KUKA KRL program: EPS_2_251491_MH05A_A_20251118025200.src

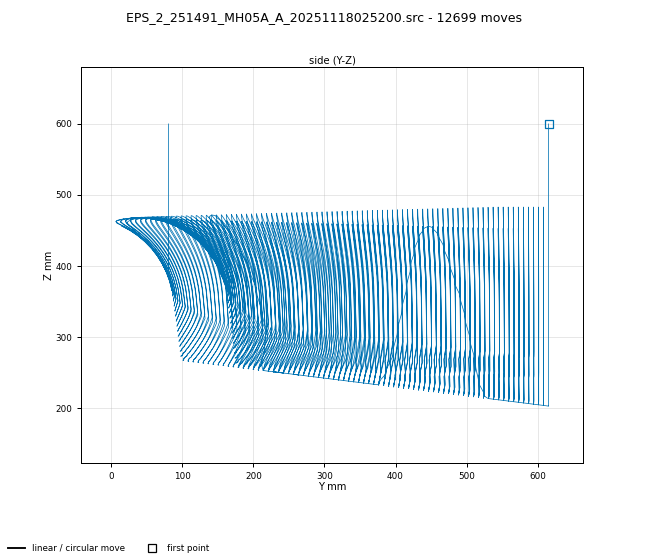
[picture p0: tool path of EPS_2_251491_MH05A_A_20251118025200.src, 12699 of 12701 moves have a stored position in this frame; points joined in program order, loops and branches not executed]
&ACCESS RVP
&REL 4
&COMMENT QRS 19112012
&PARAM EDITMASK = *
DEF PART()
EXT BAS (BAS_COMMAND :IN,REAL :IN )
INT I
BAS (#INITMOV,0 )

;KUKA QRS Post kuka4.cps  Date:22-06-2017 !

File_ID=2922

QRS_PRE_INIT()

;Init var - Until changes are made in qrs_pre_init
Outlet_Square_prg=0
Inlet_1_Square_prg=0
Inlet_2_Square_prg=0
Inlet_3_Square_prg=0
Inlet_4_Square_prg=0
Inlet_5_Square_prg=0

Outlet_1={X 0.000, Y 540.910, Z 382.500, B 0.000, E1 0.000 }
Inlet_1={X 0.000, Y 543.050, Z 352.500, B 0.000, E1 155.000 }
Outlet_1_type=201
Inlet_1_type=201
;QRS#1=Sidecore dimensions
;QRS#2=200-8" PVC SDR 35
;QRS#3=200-8" PVC SDR 35
;QRS#4=
;QRS#5=
;QRS#6=
;QRS#7=
;QRS#8=
;QRS#9=12-08 PSX
;QRS#10=12-08 PSX
;QRS#11=
;QRS#12=
;QRS#13=
;QRS#14=
;QRS#15=
;QRS#16=1220x127x762 2,5'
;QRS#17=EPS Height
;QRS#18=483
;QRS#19=*
;QRS#20= UPDATED VERSION 22-06-2017
;QRS#21=*
Outlet_Square=0100
Inlet_1_Square=0100
Inlet_2_Square=0
Inlet_3_Square=0
Inlet_4_Square=0
Inlet_5_Square=0
Mill_Square=1
Outlet_Square_Prg=204
Inlet_1_Square_prg=204

QRS_INIT()

$ADVANCE=5

; T1
PTP {E1 173.607,E2 173.607}
PTP {X 0,Y 615.506,A -85,B 0,C 180,E1 173.607,E2 173.607,E3 0,E4 0,E5 0,E6 0}
QRS_SPEED_INIT()
LIN {X 0,Y 615.506,Z 600,A -85,B 0,C 180,E1 173.607,E2 173.607,E3 0,E4 0,E5 0,E6 0} C_VEL
LIN {X 0,Y 615.506,Z 212.868,A -85,B 0,C 180,E1 173.607,E2 173.607} C_VEL
LIN {X 0,Y 615.506,Z 204.696,A -85,B 0,C 180,E1 173.607,E2 173.607} C_VEL
LIN {X 0,Y 615.486,Z 202.696,A -85,B 0,C 180,E1 173.421,E2 173.421} C_VEL
LIN {X 0,Y 615.466,Z 202.693,A -85,B 0,C 180,E1 170.801,E2 170.801} C_VEL
LIN {X 0,Y 615.486,Z 202.683,A -85,B 0,C 180,E1 168.139,E2 168.139} C_VEL
LIN {X 0,Y 615.489,Z 202.697,A -85,B 0,C 180,E1 165.451,E2 165.451} C_VEL
LIN {X 0,Y 615.458,Z 202.692,A -85,B 0,C 180,E1 162.729,E2 162.729} C_VEL
LIN {X 0,Y 615.489,Z 202.685,A -85,B 0,C 180,E1 159.967,E2 159.967} C_VEL
LIN {X 0,Y 615.474,Z 202.697,A -85,B 0,C 180,E1 157.155,E2 157.155} C_VEL
LIN {X 0,Y 615.46,Z 202.688,A -85,B 0,C 180,E1 154.436,E2 154.436} C_VEL
LIN {X 0,Y 615.493,Z 202.698,A -85,B 0,C 180,E1 151.548,E2 151.548} C_VEL
LIN {X 0,Y 615.453,Z 202.694,A -85,B 0,C 180,E1 148.919,E2 148.919} C_VEL
LIN {X 0,Y 615.455,Z 202.689,A -85,B 0,C 180,E1 146.47,E2 146.47} C_VEL
LIN {X 0,Y 615.485,Z 202.701,A -85,B 0,C 180,E1 143.575,E2 143.575} C_VEL
LIN {X 0,Y 615.448,Z 202.694,A -85,B 0,C 180,E1 140.942,E2 140.942} C_VEL
LIN {X 0,Y 615.45,Z 202.691,A -85,B 0,C 180,E1 138.523,E2 138.523} C_VEL
LIN {X 0,Y 615.494,Z 202.692,A -85,B 0,C 180,E1 135.851,E2 135.851} C_VEL
LIN {X 0,Y 615.475,Z 202.799,A -85,B 0,C 180,E1 134.199,E2 134.199} C_VEL
LIN {X 0,Y 615.458,Z 220.552,A -85,B 0,C 180,E1 131.282,E2 131.282} C_VEL
LIN {X 0,Y 615.437,Z 235.196,A -85,B 0,C 180,E1 128.908,E2 128.908} C_VEL
LIN {X 0,Y 615.496,Z 241.943,A -85,B 0,C 180,E1 127.817,E2 127.817} C_VEL
LIN {X 0,Y 615.443,Z 348.397,A -85,B 0,C 180,E1 126.553,E2 126.553} C_VEL
LIN {X 0,Y 615.464,Z 361.176,A -85,B 0,C 180,E1 126.278,E2 126.278} C_VEL
LIN {X 0,Y 615.498,Z 372.847,A -85,B 0,C 180,E1 125.908,E2 125.908} C_VEL
LIN {X 0,Y 615.47,Z 385.467,A -85,B 0,C 180,E1 125.366,E2 125.366} C_VEL
LIN {X 0,Y 615.47,Z 397.289,A -85,B 0,C 180,E1 124.698,E2 124.698} C_VEL
LIN {X 0,Y 615.497,Z 408.415,A -85,B 0,C 180,E1 123.899,E2 123.899} C_VEL
LIN {X 0,Y 615.497,Z 418.039,A -85,B 0,C 180,E1 123.04,E2 123.04} C_VEL
LIN {X 0,Y 615.496,Z 427.301,A -85,B 0,C 180,E1 122.008,E2 122.008} C_VEL
LIN {X 0,Y 615.495,Z 433.964,A -85,B 0,C 180,E1 121.087,E2 121.087} C_VEL
LIN {X 0,Y 615.499,Z 439.406,A -85,B 0,C 180,E1 120.159,E2 120.159} C_VEL
LIN {X 0,Y 615.497,Z 444.591,A -85,B 0,C 180,E1 119.031,E2 119.031} C_VEL
LIN {X 0,Y 615.492,Z 448.32,A -85,B 0,C 180,E1 117.915,E2 117.915} C_VEL
LIN {X 0,Y 615.499,Z 450.383,A -85,B 0,C 180,E1 117.046,E2 117.046} C_VEL
LIN {X 0,Y 615.495,Z 451.368,A -85,B 0,C 180,E1 116.444,E2 116.444} C_VEL
LIN {X 0,Y 615.496,Z 452.202,A -85,B 0,C 180,E1 115.57,E2 115.57} C_VEL
LIN {X 0,Y 615.496,Z 452.385,A -85,B 0,C 180,E1 114.991,E2 114.991} C_VEL
LIN {X 0,Y 615.496,Z 451.968,A -85,B 0,C 180,E1 114.009,E2 114.009} C_VEL
LIN {X 0,Y 615.494,Z 450.344,A -85,B 0,C 180,E1 112.844,E2 112.844} C_VEL
LIN {X 0,Y 615.496,Z 447.723,A -85,B 0,C 180,E1 111.783,E2 111.783} C_VEL
LIN {X 0,Y 615.497,Z 443.247,A -85,B 0,C 180,E1 110.558,E2 110.558} C_VEL
LIN {X 0,Y 615.495,Z 437.135,A -85,B 0,C 180,E1 109.338,E2 109.338} C_VEL
LIN {X 0,Y 615.498,Z 430.192,A -85,B 0,C 180,E1 108.281,E2 108.281} C_VEL
LIN {X 0,Y 615.498,Z 421.883,A -85,B 0,C 180,E1 107.27,E2 107.27} C_VEL
LIN {X 0,Y 615.497,Z 413.422,A -85,B 0,C 180,E1 106.433,E2 106.433} C_VEL
LIN {X 0,Y 615.495,Z 403.695,A -85,B 0,C 180,E1 105.65,E2 105.65} C_VEL
LIN {X 0,Y 615.46,Z 393.363,A -85,B 0,C 180,E1 104.973,E2 104.973} C_VEL
LIN {X 0,Y 615.476,Z 382.334,A -85,B 0,C 180,E1 104.395,E2 104.395} C_VEL
LIN {X 0,Y 615.49,Z 370.965,A -85,B 0,C 180,E1 103.932,E2 103.932} C_VEL
LIN {X 0,Y 615.448,Z 359.278,A -85,B 0,C 180,E1 103.58,E2 103.58} C_VEL
LIN {X 0,Y 615.432,Z 346.392,A -85,B 0,C 180,E1 103.328,E2 103.328} C_VEL
LIN {X 0,Y 615.495,Z 241.928,A -85,B 0,C 180,E1 102.091,E2 102.091} C_VEL
LIN {X 0,Y 615.436,Z 225.089,A -85,B 0,C 180,E1 99.365,E2 99.365} C_VEL
LIN {X 0,Y 615.432,Z 210.936,A -85,B 0,C 180,E1 97.052,E2 97.052} C_VEL
LIN {X 0,Y 615.459,Z 202.692,A -85,B 0,C 180,E1 95.673,E2 95.673} C_VEL
LIN {X 0,Y 615.436,Z 202.694,A -85,B 0,C 180,E1 93.273,E2 93.273} C_VEL
LIN {X 0,Y 615.438,Z 202.693,A -85,B 0,C 180,E1 91.309,E2 91.309} C_VEL
LIN {X 0,Y 615.457,Z 202.698,A -85,B 0,C 180,E1 88.691,E2 88.691} C_VEL
LIN {X 0,Y 615.491,Z 202.692,A -85,B 0,C 180,E1 86.072,E2 86.072} C_VEL
LIN {X 0,Y 615.446,Z 202.692,A -85,B 0,C 180,E1 83.443,E2 83.443} C_VEL
LIN {X 0,Y 615.447,Z 202.691,A -85,B 0,C 180,E1 81.463,E2 81.463} C_VEL
LIN {X 0,Y 615.443,Z 202.694,A -85,B 0,C 180,E1 79.135,E2 79.135} C_VEL
LIN {X 0,Y 615.459,Z 202.697,A -85,B 0,C 180,E1 76.798,E2 76.798} C_VEL
LIN {X 0,Y 615.494,Z 202.689,A -85,B 0,C 180,E1 74.095,E2 74.095} C_VEL
LIN {X 0,Y 615.448,Z 202.691,A -85,B 0,C 180,E1 71.353,E2 71.353} C_VEL
LIN {X 0,Y 615.49,Z 202.699,A -85,B 0,C 180,E1 68.568,E2 68.568} C_VEL
LIN {X 0,Y 615.47,Z 202.687,A -85,B 0,C 180,E1 65.728,E2 65.728} C_VEL
LIN {X 0,Y 615.458,Z 202.689,A -85,B 0,C 180,E1 63.555,E2 63.555} C_VEL
LIN {X 0,Y 615.45,Z 202.691,A -85,B 0,C 180,E1 61.34,E2 61.34} C_VEL
LIN {X 0,Y 615.465,Z 202.696,A -85,B 0,C 180,E1 58.918,E2 58.918} C_VEL
LIN {X 0,Y 615.492,Z 202.684,A -85,B 0,C 180,E1 55.979,E2 55.979} C_VEL
LIN {X 0,Y 615.461,Z 202.688,A -85,B 0,C 180,E1 53.574,E2 53.574} C_VEL
LIN {X 0,Y 615.469,Z 202.696,A -85,B 0,C 180,E1 50.94,E2 50.94} C_VEL
LIN {X 0,Y 615.495,Z 202.697,A -85,B 0,C 180,E1 48.527,E2 48.527} C_VEL
LIN {X 0,Y 615.484,Z 202.684,A -85,B 0,C 180,E1 45.851,E2 45.851} C_VEL
LIN {X 0,Y 615.468,Z 202.695,A -85,B 0,C 180,E1 43.046,E2 43.046} C_VEL
LIN {X 0,Y 615.495,Z 202.684,A -85,B 0,C 180,E1 40.09,E2 40.09} C_VEL
LIN {X 0,Y 615.463,Z 202.692,A -85,B 0,C 180,E1 37.244,E2 37.244} C_VEL
LIN {X 0,Y 615.491,Z 202.701,A -85,B 0,C 180,E1 34.702,E2 34.702} C_VEL
LIN {X 0,Y 615.473,Z 202.685,A -85,B 0,C 180,E1 31.686,E2 31.686} C_VEL
LIN {X 0,Y 615.465,Z 202.69,A -85,B 0,C 180,E1 29.408,E2 29.408} C_VEL
LIN {X 0,Y 615.478,Z 202.696,A -85,B 0,C 180,E1 27.044,E2 27.044} C_VEL
LIN {X 0,Y 615.486,Z 202.687,A -85,B 0,C 180,E1 24.272,E2 24.272} C_VEL
LIN {X 0,Y 615.469,Z 202.69,A -85,B 0,C 180,E1 21.433,E2 21.433} C_VEL
LIN {X 0,Y 615.484,Z 202.695,A -85,B 0,C 180,E1 18.605,E2 18.605} C_VEL
LIN {X 0,Y 615.486,Z 202.682,A -85,B 0,C 180,E1 15.905,E2 15.905} C_VEL
LIN {X 0,Y 615.477,Z 202.694,A -85,B 0,C 180,E1 13.202,E2 13.202} C_VEL
LIN {X 0,Y 615.481,Z 202.691,A -85,B 0,C 180,E1 10.527,E2 10.527} C_VEL
LIN {X 0,Y 615.487,Z 202.682,A -85,B 0,C 180,E1 7.876,E2 7.876} C_VEL
LIN {X 0,Y 615.48,Z 202.694,A -85,B 0,C 180,E1 5.241,E2 5.241} C_VEL
LIN {X 0,Y 615.48,Z 202.693,A -85,B 0,C 180,E1 2.618,E2 2.618} C_VEL
LIN {X 0,Y 615.486,Z 202.682,A -85,B 0,C 180,E1 0,E2 0} C_VEL
LIN {X 0,Y 615.479,Z 202.692,A -85,B 0,C 180,E1 -2.618,E2 -2.618} C_VEL
LIN {X 0,Y 615.481,Z 202.695,A -85,B 0,C 180,E1 -5.241,E2 -5.241} C_VEL
LIN {X 0,Y 615.487,Z 202.682,A -85,B 0,C 180,E1 -7.876,E2 -7.876} C_VEL
LIN {X 0,Y 615.48,Z 202.691,A -85,B 0,C 180,E1 -10.527,E2 -10.527} C_VEL
LIN {X 0,Y 615.479,Z 202.695,A -85,B 0,C 180,E1 -13.201,E2 -13.201} C_VEL
LIN {X 0,Y 615.486,Z 202.682,A -85,B 0,C 180,E1 -15.905,E2 -15.905} C_VEL
LIN {X 0,Y 615.486,Z 202.695,A -85,B 0,C 180,E1 -18.646,E2 -18.646} C_VEL
LIN {X 0,Y 615.47,Z 202.69,A -85,B 0,C 180,E1 -21.433,E2 -21.433} C_VEL
LIN {X 0,Y 615.485,Z 202.687,A -85,B 0,C 180,E1 -24.272,E2 -24.272} C_VEL
LIN {X 0,Y 615.473,Z 202.694,A -85,B 0,C 180,E1 -27.178,E2 -27.178} C_VEL
LIN {X 0,Y 615.481,Z 202.683,A -85,B 0,C 180,E1 -29.794,E2 -29.794} C_VEL
LIN {X 0,Y 615.486,Z 202.692,A -85,B 0,C 180,E1 -32.458,E2 -32.458} C_VEL
LIN {X 0,Y 615.494,Z 202.699,A -85,B 0,C 180,E1 -34.815,E2 -34.815} C_VEL
LIN {X 0,Y 615.465,Z 202.692,A -85,B 0,C 180,E1 -37.244,E2 -37.244} C_VEL
LIN {X 0,Y 615.495,Z 202.683,A -85,B 0,C 180,E1 -40.09,E2 -40.09} C_VEL
LIN {X 0,Y 615.47,Z 202.695,A -85,B 0,C 180,E1 -43.046,E2 -43.046} C_VEL
LIN {X 0,Y 615.484,Z 202.683,A -85,B 0,C 180,E1 -45.851,E2 -45.851} C_VEL
LIN {X 0,Y 615.49,Z 202.697,A -85,B 0,C 180,E1 -48.527,E2 -48.527} C_VEL
LIN {X 0,Y 615.462,Z 202.694,A -85,B 0,C 180,E1 -51.094,E2 -51.094} C_VEL
LIN {X 0,Y 615.463,Z 202.688,A -85,B 0,C 180,E1 -53.574,E2 -53.574} C_VEL
LIN {X 0,Y 615.49,Z 202.697,A -85,B 0,C 180,E1 -56.466,E2 -56.466} C_VEL
LIN {X 0,Y 615.458,Z 202.694,A -85,B 0,C 180,E1 -59.079,E2 -59.079} C_VEL
LIN {X 0,Y 615.46,Z 202.688,A -85,B 0,C 180,E1 -61.555,E2 -61.555} C_VEL
LIN {X 0,Y 615.495,Z 202.697,A -85,B 0,C 180,E1 -64.43,E2 -64.43} C_VEL
LIN {X 0,Y 615.451,Z 202.693,A -85,B 0,C 180,E1 -67.154,E2 -67.154} C_VEL
LIN {X 0,Y 615.481,Z 202.766,A -85,B 0,C 180,E1 -67.838,E2 -67.838} C_VEL
LIN {X 0,Y 615.467,Z 223.079,A -85,B 0,C 180,E1 -70.662,E2 -70.662} C_VEL
LIN {X 0,Y 615.458,Z 241.932,A -85,B 0,C 180,E1 -73.242,E2 -73.242} C_VEL
LIN {X 0,Y 615.495,Z 263.272,A -85,B 0,C 180,E1 -76.126,E2 -76.126} C_VEL
LIN {X 0,Y 615.46,Z 270.646,A -85,B 0,C 180,E1 -77.113,E2 -77.113} C_VEL
LIN {X 0,Y 615.467,Z 378.845,A -85,B 0,C 180,E1 -78.41,E2 -78.41} C_VEL
LIN {X 0,Y 615.463,Z 391.355,A -85,B 0,C 180,E1 -78.682,E2 -78.682} C_VEL
LIN {X 0,Y 615.484,Z 404.665,A -85,B 0,C 180,E1 -79.115,E2 -79.115} C_VEL
LIN {X 0,Y 615.486,Z 416.481,A -85,B 0,C 180,E1 -79.64,E2 -79.64} C_VEL
LIN {X 0,Y 615.492,Z 427.997,A -85,B 0,C 180,E1 -80.304,E2 -80.304} C_VEL
LIN {X 0,Y 615.499,Z 438.343,A -85,B 0,C 180,E1 -81.05,E2 -81.05} C_VEL
LIN {X 0,Y 615.497,Z 446.813,A -85,B 0,C 180,E1 -81.794,E2 -81.794} C_VEL
LIN {X 0,Y 615.498,Z 454.607,A -85,B 0,C 180,E1 -82.62,E2 -82.62} C_VEL
LIN {X 0,Y 615.496,Z 462.204,A -85,B 0,C 180,E1 -83.608,E2 -83.608} C_VEL
LIN {X 0,Y 615.498,Z 469.205,A -85,B 0,C 180,E1 -84.759,E2 -84.759} C_VEL
LIN {X 0,Y 615.494,Z 473.852,A -85,B 0,C 180,E1 -85.744,E2 -85.744} C_VEL
LIN {X 0,Y 615.494,Z 477.399,A -85,B 0,C 180,E1 -86.727,E2 -86.727} C_VEL
LIN {X 0,Y 615.497,Z 479.233,A -85,B 0,C 180,E1 -87.382,E2 -87.382} C_VEL
LIN {X 0,Y 615.499,Z 480.608,A -85,B 0,C 180,E1 -88.037,E2 -88.037} C_VEL
LIN {X 0,Y 615.496,Z 482.174,A -85,B 0,C 180,E1 -89.346,E2 -89.346} C_VEL
LIN {X 0,Y 615.494,Z 482.389,A -85,B 0,C 180,E1 -90,E2 -90} C_VEL
LIN {X 0,Y 615.495,Z 481.58,A -85,B 0,C 180,E1 -91.309,E2 -91.309} C_VEL
LIN {X 0,Y 615.499,Z 480.608,A -85,B 0,C 180,E1 -91.963,E2 -91.963} C_VEL
LIN {X 0,Y 615.497,Z 479.233,A -85,B 0,C 180,E1 -92.618,E2 -92.618} C_VEL
LIN {X 0,Y 615.496,Z 476.349,A -85,B 0,C 180,E1 -93.601,E2 -93.601} C_VEL
LIN {X 0,Y 615.498,Z 472.441,A -85,B 0,C 180,E1 -94.585,E2 -94.585} C_VEL
LIN {X 0,Y 615.499,Z 467.404,A -85,B 0,C 180,E1 -95.57,E2 -95.57} C_VEL
LIN {X 0,Y 615.497,Z 460.869,A -85,B 0,C 180,E1 -96.583,E2 -96.583} C_VEL
LIN {X 0,Y 615.497,Z 453.133,A -85,B 0,C 180,E1 -97.545,E2 -97.545} C_VEL
LIN {X 0,Y 615.498,Z 445.044,A -85,B 0,C 180,E1 -98.371,E2 -98.371} C_VEL
LIN {X 0,Y 615.499,Z 435.167,A -85,B 0,C 180,E1 -99.199,E2 -99.199} C_VEL
LIN {X 0,Y 615.491,Z 423.98,A -85,B 0,C 180,E1 -99.945,E2 -99.945} C_VEL
LIN {X 0,Y 615.487,Z 413.022,A -85,B 0,C 180,E1 -100.527,E2 -100.527} C_VEL
LIN {X 0,Y 615.473,Z 400.516,A -85,B 0,C 180,E1 -101.039,E2 -101.039} C_VEL
LIN {X 0,Y 615.463,Z 388.069,A -85,B 0,C 180,E1 -101.402,E2 -101.402} C_VEL
LIN {X 0,Y 615.47,Z 374.469,A -85,B 0,C 180,E1 -101.652,E2 -101.652} C_VEL
LIN {X 0,Y 615.46,Z 270.645,A -85,B 0,C 180,E1 -102.887,E2 -102.887} C_VEL
LIN {X 0,Y 615.465,Z 250.722,A -85,B 0,C 180,E1 -105.566,E2 -105.566} C_VEL
LIN {X 0,Y 615.484,Z 229.594,A -85,B 0,C 180,E1 -108.442,E2 -108.442} C_VEL
LIN {X 0,Y 615.476,Z 209.239,A -85,B 0,C 180,E1 -111.257,E2 -111.257} C_VEL
LIN {X 0,Y 615.478,Z 202.686,A -85,B 0,C 180,E1 -112.187,E2 -112.187} C_VEL
LIN {X 0,Y 615.471,Z 202.687,A -85,B 0,C 180,E1 -114.273,E2 -114.273} C_VEL
LIN {X 0,Y 615.46,Z 202.689,A -85,B 0,C 180,E1 -116.445,E2 -116.445} C_VEL
LIN {X 0,Y 615.454,Z 202.691,A -85,B 0,C 180,E1 -118.66,E2 -118.66} C_VEL
LIN {X 0,Y 615.47,Z 202.696,A -85,B 0,C 180,E1 -121.083,E2 -121.083} C_VEL
LIN {X 0,Y 615.492,Z 202.683,A -85,B 0,C 180,E1 -124.022,E2 -124.022} C_VEL
LIN {X 0,Y 615.464,Z 202.688,A -85,B 0,C 180,E1 -126.426,E2 -126.426} C_VEL
LIN {X 0,Y 615.472,Z 202.697,A -85,B 0,C 180,E1 -129.06,E2 -129.06} C_VEL
LIN {X 0,Y 615.491,Z 202.695,A -85,B 0,C 180,E1 -131.473,E2 -131.473} C_VEL
LIN {X 0,Y 615.485,Z 202.683,A -85,B 0,C 180,E1 -134.15,E2 -134.15} C_VEL
LIN {X 0,Y 615.475,Z 202.696,A -85,B 0,C 180,E1 -136.954,E2 -136.954} C_VEL
LIN {X 0,Y 615.494,Z 202.682,A -85,B 0,C 180,E1 -139.91,E2 -139.91} C_VEL
LIN {X 0,Y 615.47,Z 202.693,A -85,B 0,C 180,E1 -142.756,E2 -142.756} C_VEL
LIN {X 0,Y 615.491,Z 202.697,A -85,B 0,C 180,E1 -145.299,E2 -145.299} C_VEL
LIN {X 0,Y 615.481,Z 202.688,A -85,B 0,C 180,E1 -147.67,E2 -147.67} C_VEL
LIN {X 0,Y 615.483,Z 202.683,A -85,B 0,C 180,E1 -150.206,E2 -150.206} C_VEL
LIN {X 0,Y 615.489,Z 202.698,A -85,B 0,C 180,E1 -152.954,E2 -152.954} C_VEL
LIN {X 0,Y 615.483,Z 202.685,A -85,B 0,C 180,E1 -155.728,E2 -155.728} C_VEL
LIN {X 0,Y 615.476,Z 202.691,A -85,B 0,C 180,E1 -158.568,E2 -158.568} C_VEL
LIN {X 0,Y 615.478,Z 202.692,A -85,B 0,C 180,E1 -161.397,E2 -161.397} C_VEL
LIN {X 0,Y 615.487,Z 202.682,A -85,B 0,C 180,E1 -164.095,E2 -164.095} C_VEL
LIN {X 0,Y 615.487,Z 202.697,A -85,B 0,C 180,E1 -166.799,E2 -166.799} C_VEL
LIN {X 0,Y 615.473,Z 202.69,A -85,B 0,C 180,E1 -169.473,E2 -169.473} C_VEL
LIN {X 0,Y 615.489,Z 202.683,A -85,B 0,C 180,E1 -172.124,E2 -172.124} C_VEL
LIN {X 0,Y 615.488,Z 202.698,A -85,B 0,C 180,E1 -174.759,E2 -174.759} C_VEL
LIN {X 0,Y 615.469,Z 202.691,A -85,B 0,C 180,E1 -177.382,E2 -177.382} C_VEL
LIN {X 0,Y 615.486,Z 202.683,A -85,B 0,C 180,E1 -180,E2 -180} C_VEL
LIN {X 0,Y 615.487,Z 202.696,A -85,B 0,C 180,E1 -182.618,E2 -182.618} C_VEL
LIN {X 0,Y 615.468,Z 202.693,A -85,B 0,C 180,E1 -185.241,E2 -185.241} C_VEL
LIN {X 0,Y 615.486,Z 202.696,A -85,B 0,C 180,E1 -186.579,E2 -186.579} C_VEL
LIN {X 0,Y 614.796,Z 202.84,A -85,B 0,C 180,E1 -187.125,E2 -187.125} C_VEL
LIN {X 0,Y 611.95,Z 203.252,A -85,B 0,C 180,E1 -188.011,E2 -188.011} C_VEL
LIN {X 0,Y 609.561,Z 203.563,A -85,B 0,C 180,E1 -188.724,E2 -188.724} C_VEL
LIN {X 0,Y 608.533,Z 203.68,A -85,B 0,C 180,E1 -189.273,E2 -189.273} C_VEL
LIN {X 0,Y 608.447,Z 203.689,A -85,B 0,C 180,E1 -189.46,E2 -189.46} C_VEL
LIN {X 0,Y 608.462,Z 203.687,A -85,B 0,C 180,E1 -192,E2 -192} C_VEL
LIN {X 0,Y 608.47,Z 203.695,A -85,B 0,C 180,E1 -194.721,E2 -194.721} C_VEL
LIN {X 0,Y 608.437,Z 203.69,A -85,B 0,C 180,E1 -197.477,E2 -197.477} C_VEL
LIN {X 0,Y 608.436,Z 203.689,A -85,B 0,C 180,E1 -199.571,E2 -199.571} C_VEL
LIN {X 0,Y 608.476,Z 203.691,A -85,B 0,C 180,E1 -202.405,E2 -202.405} C_VEL
LIN {X 0,Y 608.447,Z 203.699,A -85,B 0,C 180,E1 -204.571,E2 -204.571} C_VEL
LIN {X 0,Y 608.433,Z 203.691,A -85,B 0,C 180,E1 -207.199,E2 -207.199} C_VEL
LIN {X 0,Y 608.462,Z 203.687,A -85,B 0,C 180,E1 -209.78,E2 -209.78} C_VEL
LIN {X 0,Y 608.465,Z 203.697,A -85,B 0,C 180,E1 -212.523,E2 -212.523} C_VEL
LIN {X 0,Y 608.422,Z 203.692,A -85,B 0,C 180,E1 -215.279,E2 -215.279} C_VEL
LIN {X 0,Y 608.465,Z 203.693,A -85,B 0,C 180,E1 -218.24,E2 -218.24} C_VEL
LIN {X 0,Y 608.415,Z 203.693,A -85,B 0,C 180,E1 -221.18,E2 -221.18} C_VEL
LIN {X 0,Y 608.465,Z 203.688,A -85,B 0,C 180,E1 -223.87,E2 -223.87} C_VEL
LIN {X 0,Y 608.486,Z 203.818,A -85,B 0,C 180,E1 -225.734,E2 -225.734} C_VEL
LIN {X 0,Y 608.467,Z 221.459,A -85,B 0,C 180,E1 -228.658,E2 -228.658} C_VEL
LIN {X 0,Y 608.415,Z 236.148,A -85,B 0,C 180,E1 -231.058,E2 -231.058} C_VEL
LIN {X 0,Y 608.457,Z 242.194,A -85,B 0,C 180,E1 -232.041,E2 -232.041} C_VEL
LIN {X 0,Y 608.509,Z 348.976,A -85,B 0,C 180,E1 -233.321,E2 -233.321} C_VEL
LIN {X 0,Y 608.507,Z 362.247,A -85,B 0,C 180,E1 -233.617,E2 -233.617} C_VEL
LIN {X 0,Y 608.519,Z 374.325,A -85,B 0,C 180,E1 -234.016,E2 -234.016} C_VEL
LIN {X 0,Y 608.505,Z 385.829,A -85,B 0,C 180,E1 -234.524,E2 -234.524} C_VEL
LIN {X 0,Y 608.47,Z 397.477,A -85,B 0,C 180,E1 -235.189,E2 -235.189} C_VEL
LIN {X 0,Y 608.472,Z 407.83,A -85,B 0,C 180,E1 -235.93,E2 -235.93} C_VEL
LIN {X 0,Y 608.471,Z 416.929,A -85,B 0,C 180,E1 -236.727,E2 -236.727} C_VEL
LIN {X 0,Y 608.455,Z 425.883,A -85,B 0,C 180,E1 -237.69,E2 -237.69} C_VEL
LIN {X 0,Y 608.458,Z 433.645,A -85,B 0,C 180,E1 -238.731,E2 -238.731} C_VEL
LIN {X 0,Y 608.446,Z 439.85,A -85,B 0,C 180,E1 -239.774,E2 -239.774} C_VEL
LIN {X 0,Y 608.428,Z 445.331,A -85,B 0,C 180,E1 -240.978,E2 -240.978} C_VEL
LIN {X 0,Y 608.437,Z 449.039,A -85,B 0,C 180,E1 -242.108,E2 -242.108} C_VEL
LIN {X 0,Y 608.428,Z 451.477,A -85,B 0,C 180,E1 -243.225,E2 -243.225} C_VEL
LIN {X 0,Y 608.431,Z 452.716,A -85,B 0,C 180,E1 -244.288,E2 -244.288} C_VEL
LIN {X 0,Y 608.416,Z 452.916,A -85,B 0,C 180,E1 -245.427,E2 -245.427} C_VEL
LIN {X 0,Y 608.442,Z 452.436,A -85,B 0,C 180,E1 -246.154,E2 -246.154} C_VEL
LIN {X 0,Y 608.432,Z 451.46,A -85,B 0,C 180,E1 -246.875,E2 -246.875} C_VEL
LIN {X 0,Y 608.436,Z 450.04,A -85,B 0,C 180,E1 -247.593,E2 -247.593} C_VEL
LIN {X 0,Y 608.44,Z 446.976,A -85,B 0,C 180,E1 -248.663,E2 -248.663} C_VEL
LIN {X 0,Y 608.443,Z 442.763,A -85,B 0,C 180,E1 -249.725,E2 -249.725} C_VEL
LIN {X 0,Y 608.445,Z 436.212,A -85,B 0,C 180,E1 -250.955,E2 -250.955} C_VEL
LIN {X 0,Y 608.464,Z 429.059,A -85,B 0,C 180,E1 -252.003,E2 -252.003} C_VEL
LIN {X 0,Y 608.458,Z 421.766,A -85,B 0,C 180,E1 -252.87,E2 -252.87} C_VEL
LIN {X 0,Y 608.47,Z 412.47,A -85,B 0,C 180,E1 -253.773,E2 -253.773} C_VEL
LIN {X 0,Y 608.478,Z 402.041,A -85,B 0,C 180,E1 -254.594,E2 -254.594} C_VEL
LIN {X 0,Y 608.482,Z 391.226,A -85,B 0,C 180,E1 -255.28,E2 -255.28} C_VEL
LIN {X 0,Y 608.526,Z 379.094,A -85,B 0,C 180,E1 -255.879,E2 -255.879} C_VEL
LIN {X 0,Y 608.498,Z 366.549,A -85,B 0,C 180,E1 -256.347,E2 -256.347} C_VEL
LIN {X 0,Y 608.484,Z 353.437,A -85,B 0,C 180,E1 -256.687,E2 -256.687} C_VEL
LIN {X 0,Y 608.495,Z 337.468,A -85,B 0,C 180,E1 -256.92,E2 -256.92} C_VEL
LIN {X 0,Y 608.486,Z 242.1,A -85,B 0,C 180,E1 -258.064,E2 -258.064} C_VEL
LIN {X 0,Y 608.427,Z 225.966,A -85,B 0,C 180,E1 -260.693,E2 -260.693} C_VEL
LIN {X 0,Y 608.455,Z 211.765,A -85,B 0,C 180,E1 -263.034,E2 -263.034} C_VEL
LIN {X 0,Y 608.425,Z 203.693,A -85,B 0,C 180,E1 -264.407,E2 -264.407} C_VEL
LIN {X 0,Y 608.408,Z 203.693,A -85,B 0,C 180,E1 -266.689,E2 -266.689} C_VEL
LIN {X 0,Y 608.457,Z 203.692,A -85,B 0,C 180,E1 -269.338,E2 -269.338} C_VEL
LIN {X 0,Y 608.466,Z 203.69,A -85,B 0,C 180,E1 -271.986,E2 -271.986} C_VEL
LIN {X 0,Y 608.414,Z 203.692,A -85,B 0,C 180,E1 -274.638,E2 -274.638} C_VEL
LIN {X 0,Y 608.438,Z 203.689,A -85,B 0,C 180,E1 -276.633,E2 -276.633} C_VEL
LIN {X 0,Y 608.423,Z 203.691,A -85,B 0,C 180,E1 -278.636,E2 -278.636} C_VEL
LIN {X 0,Y 608.434,Z 203.696,A -85,B 0,C 180,E1 -281.324,E2 -281.324} C_VEL
LIN {X 0,Y 608.473,Z 203.688,A -85,B 0,C 180,E1 -284.037,E2 -284.037} C_VEL
LIN {X 0,Y 608.424,Z 203.691,A -85,B 0,C 180,E1 -286.785,E2 -286.785} C_VEL
LIN {X 0,Y 608.448,Z 203.698,A -85,B 0,C 180,E1 -289.57,E2 -289.57} C_VEL
LIN {X 0,Y 608.431,Z 203.69,A -85,B 0,C 180,E1 -292.469,E2 -292.469} C_VEL
LIN {X 0,Y 608.435,Z 203.689,A -85,B 0,C 180,E1 -294.572,E2 -294.572} C_VEL
LIN {X 0,Y 608.464,Z 203.692,A -85,B 0,C 180,E1 -297.204,E2 -297.204} C_VEL
LIN {X 0,Y 608.47,Z 203.688,A -85,B 0,C 180,E1 -299.971,E2 -299.971} C_VEL
LIN {X 0,Y 608.445,Z 203.691,A -85,B 0,C 180,E1 -302.88,E2 -302.88} C_VEL
LIN {X 0,Y 608.436,Z 203.698,A -85,B 0,C 180,E1 -305.278,E2 -305.278} C_VEL
LIN {X 0,Y 608.462,Z 203.686,A -85,B 0,C 180,E1 -308.239,E2 -308.239} C_VEL
LIN {X 0,Y 608.461,Z 203.697,A -85,B 0,C 180,E1 -311.342,E2 -311.342} C_VEL
LIN {X 0,Y 608.452,Z 203.687,A -85,B 0,C 180,E1 -314.263,E2 -314.263} C_VEL
LIN {X 0,Y 608.437,Z 203.695,A -85,B 0,C 180,E1 -317.038,E2 -317.038} C_VEL
LIN {X 0,Y 608.457,Z 203.691,A -85,B 0,C 180,E1 -319.697,E2 -319.697} C_VEL
LIN {X 0,Y 608.461,Z 203.686,A -85,B 0,C 180,E1 -322.253,E2 -322.253} C_VEL
LIN {X 0,Y 608.435,Z 203.692,A -85,B 0,C 180,E1 -324.722,E2 -324.722} C_VEL
LIN {X 0,Y 608.462,Z 203.693,A -85,B 0,C 180,E1 -327.477,E2 -327.477} C_VEL
LIN {X 0,Y 608.466,Z 203.686,A -85,B 0,C 180,E1 -330.22,E2 -330.22} C_VEL
LIN {X 0,Y 608.468,Z 203.689,A -85,B 0,C 180,E1 -332.794,E2 -332.794} C_VEL
LIN {X 0,Y 608.452,Z 203.694,A -85,B 0,C 180,E1 -335.429,E2 -335.429} C_VEL
LIN {X 0,Y 608.461,Z 203.686,A -85,B 0,C 180,E1 -338.308,E2 -338.308} C_VEL
LIN {X 0,Y 608.451,Z 203.698,A -85,B 0,C 180,E1 -341.13,E2 -341.13} C_VEL
LIN {X 0,Y 608.459,Z 203.687,A -85,B 0,C 180,E1 -343.906,E2 -343.906} C_VEL
LIN {X 0,Y 608.458,Z 203.69,A -85,B 0,C 180,E1 -346.643,E2 -346.643} C_VEL
LIN {X 0,Y 608.462,Z 203.692,A -85,B 0,C 180,E1 -349.35,E2 -349.35} C_VEL
LIN {X 0,Y 608.477,Z 203.684,A -85,B 0,C 180,E1 -352.033,E2 -352.033} C_VEL
LIN {X 0,Y 608.46,Z 203.691,A -85,B 0,C 180,E1 -354.698,E2 -354.698} C_VEL
LIN {X 0,Y 608.471,Z 203.69,A -85,B 0,C 180,E1 -357.352,E2 -357.352} C_VEL
LIN {X 0,Y 608.477,Z 203.684,A -85,B 0,C 180,E1 -360,E2 -360} C_VEL
LIN {X 0,Y 608.47,Z 203.69,A -85,B 0,C 180,E1 -362.648,E2 -362.648} C_VEL
LIN {X 0,Y 608.462,Z 203.691,A -85,B 0,C 180,E1 -365.302,E2 -365.302} C_VEL
LIN {X 0,Y 608.477,Z 203.684,A -85,B 0,C 180,E1 -367.967,E2 -367.967} C_VEL
LIN {X 0,Y 608.467,Z 203.696,A -85,B 0,C 180,E1 -370.957,E2 -370.957} C_VEL
LIN {X 0,Y 608.459,Z 203.69,A -85,B 0,C 180,E1 -373.357,E2 -373.357} C_VEL
LIN {X 0,Y 608.459,Z 203.687,A -85,B 0,C 180,E1 -376.094,E2 -376.094} C_VEL
LIN {X 0,Y 608.452,Z 203.698,A -85,B 0,C 180,E1 -378.87,E2 -378.87} C_VEL
LIN {X 0,Y 608.461,Z 203.686,A -85,B 0,C 180,E1 -381.692,E2 -381.692} C_VEL
LIN {X 0,Y 608.452,Z 203.693,A -85,B 0,C 180,E1 -384.571,E2 -384.571} C_VEL
LIN {X 0,Y 608.469,Z 203.689,A -85,B 0,C 180,E1 -387.207,E2 -387.207} C_VEL
LIN {X 0,Y 608.466,Z 203.686,A -85,B 0,C 180,E1 -389.972,E2 -389.972} C_VEL
LIN {X 0,Y 608.449,Z 203.697,A -85,B 0,C 180,E1 -392.88,E2 -392.88} C_VEL
LIN {X 0,Y 608.437,Z 203.692,A -85,B 0,C 180,E1 -395.278,E2 -395.278} C_VEL
LIN {X 0,Y 608.467,Z 203.688,A -85,B 0,C 180,E1 -398.241,E2 -398.241} C_VEL
LIN {X 0,Y 608.436,Z 203.692,A -85,B 0,C 180,E1 -401.178,E2 -401.178} C_VEL
LIN {X 0,Y 608.467,Z 203.686,A -85,B 0,C 180,E1 -403.87,E2 -403.87} C_VEL
LIN {X 0,Y 608.478,Z 203.695,A -85,B 0,C 180,E1 -406.691,E2 -406.691} C_VEL
LIN {X 0,Y 608.448,Z 203.696,A -85,B 0,C 180,E1 -408.823,E2 -408.823} C_VEL
LIN {X 0,Y 608.461,Z 203.686,A -85,B 0,C 180,E1 -411.761,E2 -411.761} C_VEL
LIN {X 0,Y 608.447,Z 203.689,A -85,B 0,C 180,E1 -413.955,E2 -413.955} C_VEL
LIN {X 0,Y 608.467,Z 203.691,A -85,B 0,C 180,E1 -416.33,E2 -416.33} C_VEL
LIN {X 0,Y 608.443,Z 203.697,A -85,B 0,C 180,E1 -418.733,E2 -418.733} C_VEL
LIN {X 0,Y 608.448,Z 203.688,A -85,B 0,C 180,E1 -421.385,E2 -421.385} C_VEL
LIN {X 0,Y 608.476,Z 203.69,A -85,B 0,C 180,E1 -424.279,E2 -424.279} C_VEL
LIN {X 0,Y 608.434,Z 203.696,A -85,B 0,C 180,E1 -426.876,E2 -426.876} C_VEL
LIN {X 0,Y 608.474,Z 203.892,A -85,B 0,C 180,E1 -427.729,E2 -427.729} C_VEL
LIN {X 0,Y 608.549,Z 220.578,A -85,B 0,C 180,E1 -430.081,E2 -430.081} C_VEL
LIN {X 0,Y 608.477,Z 240.727,A -85,B 0,C 180,E1 -432.871,E2 -432.871} C_VEL
LIN {X 0,Y 608.5,Z 260.877,A -85,B 0,C 180,E1 -435.622,E2 -435.622} C_VEL
LIN {X 0,Y 608.467,Z 271.158,A -85,B 0,C 180,E1 -436.984,E2 -436.984} C_VEL
LIN {X 0,Y 608.531,Z 378.957,A -85,B 0,C 180,E1 -438.276,E2 -438.276} C_VEL
LIN {X 0,Y 608.498,Z 392.223,A -85,B 0,C 180,E1 -438.571,E2 -438.571} C_VEL
LIN {X 0,Y 608.51,Z 404.168,A -85,B 0,C 180,E1 -438.965,E2 -438.965} C_VEL
LIN {X 0,Y 608.504,Z 416.638,A -85,B 0,C 180,E1 -439.519,E2 -439.519} C_VEL
LIN {X 0,Y 608.483,Z 428.2,A -85,B 0,C 180,E1 -440.191,E2 -440.191} C_VEL
LIN {X 0,Y 608.485,Z 438.596,A -85,B 0,C 180,E1 -440.946,E2 -440.946} C_VEL
LIN {X 0,Y 608.475,Z 447.113,A -85,B 0,C 180,E1 -441.699,E2 -441.699} C_VEL
LIN {X 0,Y 608.471,Z 454.962,A -85,B 0,C 180,E1 -442.534,E2 -442.534} C_VEL
LIN {X 0,Y 608.461,Z 462.287,A -85,B 0,C 180,E1 -443.485,E2 -443.485} C_VEL
LIN {X 0,Y 608.45,Z 467.867,A -85,B 0,C 180,E1 -444.366,E2 -444.366} C_VEL
LIN {X 0,Y 608.432,Z 472.951,A -85,B 0,C 180,E1 -445.362,E2 -445.362} C_VEL
LIN {X 0,Y 608.449,Z 476.897,A -85,B 0,C 180,E1 -446.358,E2 -446.358} C_VEL
LIN {X 0,Y 608.425,Z 479.809,A -85,B 0,C 180,E1 -447.352,E2 -447.352} C_VEL
LIN {X 0,Y 608.444,Z 481.202,A -85,B 0,C 180,E1 -448.014,E2 -448.014} C_VEL
LIN {X 0,Y 608.438,Z 482.784,A -85,B 0,C 180,E1 -449.338,E2 -449.338} C_VEL
LIN {X 0,Y 608.434,Z 483,A -85,B 0,C 180,E1 -450,E2 -450} C_VEL
LIN {X 0,Y 608.448,Z 482.184,A -85,B 0,C 180,E1 -451.324,E2 -451.324} C_VEL
LIN {X 0,Y 608.444,Z 481.201,A -85,B 0,C 180,E1 -451.986,E2 -451.986} C_VEL
LIN {X 0,Y 608.425,Z 479.809,A -85,B 0,C 180,E1 -452.648,E2 -452.648} C_VEL
LIN {X 0,Y 608.449,Z 476.896,A -85,B 0,C 180,E1 -453.642,E2 -453.642} C_VEL
LIN {X 0,Y 608.432,Z 472.95,A -85,B 0,C 180,E1 -454.638,E2 -454.638} C_VEL
LIN {X 0,Y 608.437,Z 466.876,A -85,B 0,C 180,E1 -455.801,E2 -455.801} C_VEL
LIN {X 0,Y 608.462,Z 460.235,A -85,B 0,C 180,E1 -456.799,E2 -456.799} C_VEL
LIN {X 0,Y 608.456,Z 451.989,A -85,B 0,C 180,E1 -457.8,E2 -457.8} C_VEL
LIN {X 0,Y 608.472,Z 443.536,A -85,B 0,C 180,E1 -458.636,E2 -458.636} C_VEL
LIN {X 0,Y 608.478,Z 433.09,A -85,B 0,C 180,E1 -459.473,E2 -459.473} C_VEL
LIN {X 0,Y 608.501,Z 422.755,A -85,B 0,C 180,E1 -460.145,E2 -460.145} C_VEL
LIN {X 0,Y 608.517,Z 411.6,A -85,B 0,C 180,E1 -460.724,E2 -460.724} C_VEL
LIN {X 0,Y 608.515,Z 399.9,A -85,B 0,C 180,E1 -461.192,E2 -461.192} C_VEL
LIN {X 0,Y 608.528,Z 387.265,A -85,B 0,C 180,E1 -461.555,E2 -461.555} C_VEL
LIN {X 0,Y 608.533,Z 374.599,A -85,B 0,C 180,E1 -461.787,E2 -461.787} C_VEL
LIN {X 0,Y 608.467,Z 271.14,A -85,B 0,C 180,E1 -463.017,E2 -463.017} C_VEL
LIN {X 0,Y 608.46,Z 253.319,A -85,B 0,C 180,E1 -465.406,E2 -465.406} C_VEL
LIN {X 0,Y 608.51,Z 233.17,A -85,B 0,C 180,E1 -468.17,E2 -468.17} C_VEL
LIN {X 0,Y 608.526,Z 214.438,A -85,B 0,C 180,E1 -470.78,E2 -470.78} C_VEL
LIN {X 0,Y 608.44,Z 203.691,A -85,B 0,C 180,E1 -472.317,E2 -472.317} C_VEL
LIN {X 0,Y 608.436,Z 203.69,A -85,B 0,C 180,E1 -474.572,E2 -474.572} C_VEL
LIN {X 0,Y 608.467,Z 203.692,A -85,B 0,C 180,E1 -477.205,E2 -477.205} C_VEL
LIN {X 0,Y 608.47,Z 203.687,A -85,B 0,C 180,E1 -479.972,E2 -479.972} C_VEL
LIN {X 0,Y 608.449,Z 203.691,A -85,B 0,C 180,E1 -482.88,E2 -482.88} C_VEL
LIN {X 0,Y 608.436,Z 203.699,A -85,B 0,C 180,E1 -485.278,E2 -485.278} C_VEL
LIN {X 0,Y 608.468,Z 203.689,A -85,B 0,C 180,E1 -487.746,E2 -487.746} C_VEL
LIN {X 0,Y 608.442,Z 203.689,A -85,B 0,C 180,E1 -490.328,E2 -490.328} C_VEL
LIN {X 0,Y 608.443,Z 203.694,A -85,B 0,C 180,E1 -492.96,E2 -492.96} C_VEL
LIN {X 0,Y 608.459,Z 203.689,A -85,B 0,C 180,E1 -495.736,E2 -495.736} C_VEL
LIN {X 0,Y 608.447,Z 203.69,A -85,B 0,C 180,E1 -498.659,E2 -498.659} C_VEL
LIN {X 0,Y 608.469,Z 203.692,A -85,B 0,C 180,E1 -501.412,E2 -501.412} C_VEL
LIN {X 0,Y 608.477,Z 203.685,A -85,B 0,C 180,E1 -503.95,E2 -503.95} C_VEL
LIN {X 0,Y 608.444,Z 203.689,A -85,B 0,C 180,E1 -506.328,E2 -506.328} C_VEL
LIN {X 0,Y 608.444,Z 203.692,A -85,B 0,C 180,E1 -508.732,E2 -508.732} C_VEL
LIN {X 0,Y 608.471,Z 203.691,A -85,B 0,C 180,E1 -511.38,E2 -511.38} C_VEL
LIN {X 0,Y 608.439,Z 203.689,A -85,B 0,C 180,E1 -513.964,E2 -513.964} C_VEL
LIN {X 0,Y 608.467,Z 203.685,A -85,B 0,C 180,E1 -516.155,E2 -516.155} C_VEL
LIN {X 0,Y 608.464,Z 203.687,A -85,B 0,C 180,E1 -518.308,E2 -518.308} C_VEL
LIN {X 0,Y 608.466,Z 203.691,A -85,B 0,C 180,E1 -521.285,E2 -521.285} C_VEL
LIN {X 0,Y 608.458,Z 203.687,A -85,B 0,C 180,E1 -523.906,E2 -523.906} C_VEL
LIN {X 0,Y 608.465,Z 203.691,A -85,B 0,C 180,E1 -526.644,E2 -526.644} C_VEL
LIN {X 0,Y 608.456,Z 203.69,A -85,B 0,C 180,E1 -529.35,E2 -529.35} C_VEL
LIN {X 0,Y 608.478,Z 203.684,A -85,B 0,C 180,E1 -532.033,E2 -532.033} C_VEL
LIN {X 0,Y 608.468,Z 203.693,A -85,B 0,C 180,E1 -534.698,E2 -534.698} C_VEL
LIN {X 0,Y 608.463,Z 203.689,A -85,B 0,C 180,E1 -537.352,E2 -537.352} C_VEL
LIN {X 0,Y 608.477,Z 203.684,A -85,B 0,C 180,E1 -540,E2 -540} C_VEL
LIN {X 0,Y 608.477,Z 203.692,A -85,B 0,C 180,E1 -542.648,E2 -542.648} C_VEL
LIN {X 0,Y 608.45,Z 203.69,A -85,B 0,C 180,E1 -545.302,E2 -545.302} C_VEL
LIN {X 0,Y 608.477,Z 203.685,A -85,B 0,C 180,E1 -547.967,E2 -547.967} C_VEL
LIN {X 0,Y 608.447,Z 203.689,A -85,B 0,C 180,E1 -549.46,E2 -549.46} C_VEL
LIN {X 0,Y 607.777,Z 203.773,A -85,B 0,C 180,E1 -550.012,E2 -550.012} C_VEL
LIN {X 0,Y 604.929,Z 204.133,A -85,B 0,C 180,E1 -550.909,E2 -550.909} C_VEL
LIN {X 0,Y 602.526,Z 204.429,A -85,B 0,C 180,E1 -551.631,E2 -551.631} C_VEL
LIN {X 0,Y 601.493,Z 204.557,A -85,B 0,C 180,E1 -552.187,E2 -552.187} C_VEL
LIN {X 0,Y 601.408,Z 204.568,A -85,B 0,C 180,E1 -552.376,E2 -552.376} C_VEL
LIN {X 0,Y 601.422,Z 204.57,A -85,B 0,C 180,E1 -554.897,E2 -554.897} C_VEL
LIN {X 0,Y 601.428,Z 204.568,A -85,B 0,C 180,E1 -556.986,E2 -556.986} C_VEL
LIN {X 0,Y 601.398,Z 204.566,A -85,B 0,C 180,E1 -559.81,E2 -559.81} C_VEL
LIN {X 0,Y 601.414,Z 204.575,A -85,B 0,C 180,E1 -562.606,E2 -562.606} C_VEL
LIN {X 0,Y 601.39,Z 204.573,A -85,B 0,C 180,E1 -564.879,E2 -564.879} C_VEL
LIN {X 0,Y 601.387,Z 204.568,A -85,B 0,C 180,E1 -567.358,E2 -567.358} C_VEL
LIN {X 0,Y 601.396,Z 204.566,A -85,B 0,C 180,E1 -569.395,E2 -569.395} C_VEL
LIN {X 0,Y 601.397,Z 204.567,A -85,B 0,C 180,E1 -571.727,E2 -571.727} C_VEL
LIN {X 0,Y 601.418,Z 204.568,A -85,B 0,C 180,E1 -574.119,E2 -574.119} C_VEL
LIN {X 0,Y 601.388,Z 204.576,A -85,B 0,C 180,E1 -576.584,E2 -576.584} C_VEL
LIN {X 0,Y 601.386,Z 204.569,A -85,B 0,C 180,E1 -579.129,E2 -579.129} C_VEL
LIN {X 0,Y 601.419,Z 204.565,A -85,B 0,C 180,E1 -581.766,E2 -581.766} C_VEL
LIN {X 0,Y 601.398,Z 204.576,A -85,B 0,C 180,E1 -584.533,E2 -584.533} C_VEL
LIN {X 0,Y 601.438,Z 204.672,A -85,B 0,C 180,E1 -585.643,E2 -585.643} C_VEL
LIN {X 0,Y 601.491,Z 218.887,A -85,B 0,C 180,E1 -588.033,E2 -588.033} C_VEL
LIN {X 0,Y 601.396,Z 236.03,A -85,B 0,C 180,E1 -590.872,E2 -590.872} C_VEL
LIN {X 0,Y 601.441,Z 242.227,A -85,B 0,C 180,E1 -591.887,E2 -591.887} C_VEL
LIN {X 0,Y 601.697,Z 250.537,A -85,B 0,C 180,E1 -591.992,E2 -591.992} C_VEL
LIN {X 0,Y 601.566,Z 349.498,A -85,B 0,C 180,E1 -593.194,E2 -593.194} C_VEL
LIN {X 0,Y 601.545,Z 362.704,A -85,B 0,C 180,E1 -593.496,E2 -593.496} C_VEL
LIN {X 0,Y 601.548,Z 375.739,A -85,B 0,C 180,E1 -593.94,E2 -593.94} C_VEL
LIN {X 0,Y 601.484,Z 387.972,A -85,B 0,C 180,E1 -594.513,E2 -594.513} C_VEL
LIN {X 0,Y 601.459,Z 398.993,A -85,B 0,C 180,E1 -595.173,E2 -595.173} C_VEL
LIN {X 0,Y 601.44,Z 408.579,A -85,B 0,C 180,E1 -595.883,E2 -595.883} C_VEL
LIN {X 0,Y 601.409,Z 417.528,A -85,B 0,C 180,E1 -596.685,E2 -596.685} C_VEL
LIN {X 0,Y 601.402,Z 426.505,A -85,B 0,C 180,E1 -597.681,E2 -597.681} C_VEL
LIN {X 0,Y 601.385,Z 432.945,A -85,B 0,C 180,E1 -598.551,E2 -598.551} C_VEL
LIN {X 0,Y 601.355,Z 439.453,A -85,B 0,C 180,E1 -599.638,E2 -599.638} C_VEL
LIN {X 0,Y 601.352,Z 444.012,A -85,B 0,C 180,E1 -600.603,E2 -600.603} C_VEL
LIN {X 0,Y 601.338,Z 448.127,A -85,B 0,C 180,E1 -601.749,E2 -601.749} C_VEL
LIN {X 0,Y 601.335,Z 450.93,A -85,B 0,C 180,E1 -602.883,E2 -602.883} C_VEL
LIN {X 0,Y 601.336,Z 452.626,A -85,B 0,C 180,E1 -604.149,E2 -604.149} C_VEL
LIN {X 0,Y 601.33,Z 452.989,A -85,B 0,C 180,E1 -605.118,E2 -605.118} C_VEL
LIN {X 0,Y 601.347,Z 452.686,A -85,B 0,C 180,E1 -605.855,E2 -605.855} C_VEL
LIN {X 0,Y 601.326,Z 451.948,A -85,B 0,C 180,E1 -606.586,E2 -606.586} C_VEL
LIN {X 0,Y 601.337,Z 450.488,A -85,B 0,C 180,E1 -607.414,E2 -607.414} C_VEL
LIN {X 0,Y 601.342,Z 447.945,A -85,B 0,C 180,E1 -608.399,E2 -608.399} C_VEL
LIN {X 0,Y 601.356,Z 444.059,A -85,B 0,C 180,E1 -609.476,E2 -609.476} C_VEL
LIN {X 0,Y 601.379,Z 438.949,A -85,B 0,C 180,E1 -610.545,E2 -610.545} C_VEL
LIN {X 0,Y 601.379,Z 432.491,A -85,B 0,C 180,E1 -611.607,E2 -611.607} C_VEL
LIN {X 0,Y 601.399,Z 424.407,A -85,B 0,C 180,E1 -612.663,E2 -612.663} C_VEL
LIN {X 0,Y 601.425,Z 415.546,A -85,B 0,C 180,E1 -613.593,E2 -613.593} C_VEL
LIN {X 0,Y 601.446,Z 406.049,A -85,B 0,C 180,E1 -614.41,E2 -614.41} C_VEL
LIN {X 0,Y 601.458,Z 394.737,A -85,B 0,C 180,E1 -615.19,E2 -615.19} C_VEL
LIN {X 0,Y 601.505,Z 383.645,A -85,B 0,C 180,E1 -615.797,E2 -615.797} C_VEL
LIN {X 0,Y 601.563,Z 372.184,A -85,B 0,C 180,E1 -616.285,E2 -616.285} C_VEL
LIN {X 0,Y 601.541,Z 359.608,A -85,B 0,C 180,E1 -616.681,E2 -616.681} C_VEL
LIN {X 0,Y 601.548,Z 346.886,A -85,B 0,C 180,E1 -616.938,E2 -616.938} C_VEL
LIN {X 0,Y 601.595,Z 243.225,A -85,B 0,C 180,E1 -618.188,E2 -618.188} C_VEL
LIN {X 0,Y 601.423,Z 242.116,A -85,B 0,C 180,E1 -618.217,E2 -618.217} C_VEL
LIN {X 0,Y 601.413,Z 226.732,A -85,B 0,C 180,E1 -620.754,E2 -620.754} C_VEL
LIN {X 0,Y 601.457,Z 212.535,A -85,B 0,C 180,E1 -623.121,E2 -623.121} C_VEL
LIN {X 0,Y 601.39,Z 204.57,A -85,B 0,C 180,E1 -624.467,E2 -624.467} C_VEL
LIN {X 0,Y 601.42,Z 204.568,A -85,B 0,C 180,E1 -627.321,E2 -627.321} C_VEL
LIN {X 0,Y 601.445,Z 204.565,A -85,B 0,C 180,E1 -630,E2 -630} C_VEL
LIN {X 0,Y 601.406,Z 204.565,A -85,B 0,C 180,E1 -632.679,E2 -632.679} C_VEL
LIN {X 0,Y 601.409,Z 204.571,A -85,B 0,C 180,E1 -635.364,E2 -635.364} C_VEL
LIN {X 0,Y 601.439,Z 204.564,A -85,B 0,C 180,E1 -638.061,E2 -638.061} C_VEL
LIN {X 0,Y 601.405,Z 204.567,A -85,B 0,C 180,E1 -641,E2 -641} C_VEL
LIN {X 0,Y 601.408,Z 204.575,A -85,B 0,C 180,E1 -643.516,E2 -643.516} C_VEL
LIN {X 0,Y 601.414,Z 204.565,A -85,B 0,C 180,E1 -646.287,E2 -646.287} C_VEL
LIN {X 0,Y 601.41,Z 204.568,A -85,B 0,C 180,E1 -649.099,E2 -649.099} C_VEL
LIN {X 0,Y 601.401,Z 204.569,A -85,B 0,C 180,E1 -651.959,E2 -651.959} C_VEL
LIN {X 0,Y 601.39,Z 204.569,A -85,B 0,C 180,E1 -654.879,E2 -654.879} C_VEL
LIN {X 0,Y 601.396,Z 204.57,A -85,B 0,C 180,E1 -657.868,E2 -657.868} C_VEL
LIN {X 0,Y 601.407,Z 204.566,A -85,B 0,C 180,E1 -660.165,E2 -660.165} C_VEL
LIN {X 0,Y 601.406,Z 204.566,A -85,B 0,C 180,E1 -662.712,E2 -662.712} C_VEL
LIN {X 0,Y 601.383,Z 204.574,A -85,B 0,C 180,E1 -665.11,E2 -665.11} C_VEL
LIN {X 0,Y 601.433,Z 204.572,A -85,B 0,C 180,E1 -667.419,E2 -667.419} C_VEL
LIN {X 0,Y 601.401,Z 204.567,A -85,B 0,C 180,E1 -669.995,E2 -669.995} C_VEL
LIN {X 0,Y 601.384,Z 204.569,A -85,B 0,C 180,E1 -672.672,E2 -672.672} C_VEL
LIN {X 0,Y 601.426,Z 204.571,A -85,B 0,C 180,E1 -675.482,E2 -675.482} C_VEL
LIN {X 0,Y 601.415,Z 204.564,A -85,B 0,C 180,E1 -678.407,E2 -678.407} C_VEL
LIN {X 0,Y 601.403,Z 204.569,A -85,B 0,C 180,E1 -680.872,E2 -680.872} C_VEL
LIN {X 0,Y 601.441,Z 204.564,A -85,B 0,C 180,E1 -683.734,E2 -683.734} C_VEL
LIN {X 0,Y 601.411,Z 204.567,A -85,B 0,C 180,E1 -686.685,E2 -686.685} C_VEL
LIN {X 0,Y 601.412,Z 204.572,A -85,B 0,C 180,E1 -689.057,E2 -689.057} C_VEL
LIN {X 0,Y 601.435,Z 204.57,A -85,B 0,C 180,E1 -691.373,E2 -691.373} C_VEL
LIN {X 0,Y 601.404,Z 204.566,A -85,B 0,C 180,E1 -694.133,E2 -694.133} C_VEL
LIN {X 0,Y 601.417,Z 204.566,A -85,B 0,C 180,E1 -696.589,E2 -696.589} C_VEL
LIN {X 0,Y 601.431,Z 204.567,A -85,B 0,C 180,E1 -699.478,E2 -699.478} C_VEL
LIN {X 0,Y 601.393,Z 204.567,A -85,B 0,C 180,E1 -702.311,E2 -702.311} C_VEL
LIN {X 0,Y 601.409,Z 204.566,A -85,B 0,C 180,E1 -704.408,E2 -704.408} C_VEL
LIN {X 0,Y 601.414,Z 204.574,A -85,B 0,C 180,E1 -707.172,E2 -707.172} C_VEL
LIN {X 0,Y 601.433,Z 204.562,A -85,B 0,C 180,E1 -709.905,E2 -709.905} C_VEL
LIN {X 0,Y 601.437,Z 204.565,A -85,B 0,C 180,E1 -712.615,E2 -712.615} C_VEL
LIN {X 0,Y 601.415,Z 204.57,A -85,B 0,C 180,E1 -715.308,E2 -715.308} C_VEL
LIN {X 0,Y 601.435,Z 204.562,A -85,B 0,C 180,E1 -717.991,E2 -717.991} C_VEL
LIN {X 0,Y 601.442,Z 204.566,A -85,B 0,C 180,E1 -720.669,E2 -720.669} C_VEL
LIN {X 0,Y 601.426,Z 204.567,A -85,B 0,C 180,E1 -723.35,E2 -723.35} C_VEL
LIN {X 0,Y 601.435,Z 204.562,A -85,B 0,C 180,E1 -726.037,E2 -726.037} C_VEL
LIN {X 0,Y 601.41,Z 204.572,A -85,B 0,C 180,E1 -728.738,E2 -728.738} C_VEL
LIN {X 0,Y 601.432,Z 204.564,A -85,B 0,C 180,E1 -731.458,E2 -731.458} C_VEL
LIN {X 0,Y 601.417,Z 204.565,A -85,B 0,C 180,E1 -734.206,E2 -734.206} C_VEL
LIN {X 0,Y 601.428,Z 204.572,A -85,B 0,C 180,E1 -736.986,E2 -736.986} C_VEL
LIN {X 0,Y 601.402,Z 204.566,A -85,B 0,C 180,E1 -739.81,E2 -739.81} C_VEL
LIN {X 0,Y 601.413,Z 204.571,A -85,B 0,C 180,E1 -742.606,E2 -742.606} C_VEL
LIN {X 0,Y 601.398,Z 204.576,A -85,B 0,C 180,E1 -744.879,E2 -744.879} C_VEL
LIN {X 0,Y 601.409,Z 204.567,A -85,B 0,C 180,E1 -747.362,E2 -747.362} C_VEL
LIN {X 0,Y 601.426,Z 204.564,A -85,B 0,C 180,E1 -750.164,E2 -750.164} C_VEL
LIN {X 0,Y 601.418,Z 204.574,A -85,B 0,C 180,E1 -752.716,E2 -752.716} C_VEL
LIN {X 0,Y 601.398,Z 204.571,A -85,B 0,C 180,E1 -755.113,E2 -755.113} C_VEL
LIN {X 0,Y 601.43,Z 204.563,A -85,B 0,C 180,E1 -757.42,E2 -757.42} C_VEL
LIN {X 0,Y 601.401,Z 204.567,A -85,B 0,C 180,E1 -759.996,E2 -759.996} C_VEL
LIN {X 0,Y 601.407,Z 204.575,A -85,B 0,C 180,E1 -762.671,E2 -762.671} C_VEL
LIN {X 0,Y 601.397,Z 204.567,A -85,B 0,C 180,E1 -765.48,E2 -765.48} C_VEL
LIN {X 0,Y 601.424,Z 204.566,A -85,B 0,C 180,E1 -768.235,E2 -768.235} C_VEL
LIN {X 0,Y 601.402,Z 204.572,A -85,B 0,C 180,E1 -770.873,E2 -770.873} C_VEL
LIN {X 0,Y 601.391,Z 204.567,A -85,B 0,C 180,E1 -773.417,E2 -773.417} C_VEL
LIN {X 0,Y 601.432,Z 204.564,A -85,B 0,C 180,E1 -776.065,E2 -776.065} C_VEL
LIN {X 0,Y 601.399,Z 204.569,A -85,B 0,C 180,E1 -779.057,E2 -779.057} C_VEL
LIN {X 0,Y 601.408,Z 204.565,A -85,B 0,C 180,E1 -781.372,E2 -781.372} C_VEL
LIN {X 0,Y 601.41,Z 204.569,A -85,B 0,C 180,E1 -784.134,E2 -784.134} C_VEL
LIN {X 0,Y 601.393,Z 204.578,A -85,B 0,C 180,E1 -786.589,E2 -786.589} C_VEL
LIN {X 0,Y 601.402,Z 204.618,A -85,B 0,C 180,E1 -787.557,E2 -787.557} C_VEL
LIN {X 0,Y 601.664,Z 210.504,A -85,B 0,C 180,E1 -788.411,E2 -788.411} C_VEL
LIN {X 0,Y 601.56,Z 229.815,A -85,B 0,C 180,E1 -791.142,E2 -791.142} C_VEL
LIN {X 0,Y 601.493,Z 249.543,A -85,B 0,C 180,E1 -793.889,E2 -793.889} C_VEL
LIN {X 0,Y 601.463,Z 270.322,A -85,B 0,C 180,E1 -796.743,E2 -796.743} C_VEL
LIN {X 0,Y 601.448,Z 271.158,A -85,B 0,C 180,E1 -796.829,E2 -796.829} C_VEL
LIN {X 0,Y 601.639,Z 331.974,A -85,B 0,C 180,E1 -797.563,E2 -797.563} C_VEL
LIN {X 0,Y 601.602,Z 378.957,A -85,B 0,C 180,E1 -798.14,E2 -798.14} C_VEL
LIN {X 0,Y 601.562,Z 392.224,A -85,B 0,C 180,E1 -798.438,E2 -798.438} C_VEL
LIN {X 0,Y 601.534,Z 404,A -85,B 0,C 180,E1 -798.829,E2 -798.829} C_VEL
LIN {X 0,Y 601.526,Z 414.928,A -85,B 0,C 180,E1 -799.311,E2 -799.311} C_VEL
LIN {X 0,Y 601.484,Z 425.584,A -85,B 0,C 180,E1 -799.906,E2 -799.906} C_VEL
LIN {X 0,Y 601.448,Z 436.478,A -85,B 0,C 180,E1 -800.67,E2 -800.67} C_VEL
LIN {X 0,Y 601.429,Z 447.114,A -85,B 0,C 180,E1 -801.601,E2 -801.601} C_VEL
LIN {X 0,Y 601.418,Z 454.962,A -85,B 0,C 180,E1 -802.446,E2 -802.446} C_VEL
LIN {X 0,Y 601.37,Z 462.225,A -85,B 0,C 180,E1 -803.398,E2 -803.398} C_VEL
LIN {X 0,Y 601.372,Z 467.867,A -85,B 0,C 180,E1 -804.299,E2 -804.299} C_VEL
LIN {X 0,Y 601.336,Z 472.951,A -85,B 0,C 180,E1 -805.307,E2 -805.307} C_VEL
LIN {X 0,Y 601.368,Z 476.896,A -85,B 0,C 180,E1 -806.315,E2 -806.315} C_VEL
LIN {X 0,Y 601.325,Z 479.809,A -85,B 0,C 180,E1 -807.321,E2 -807.321} C_VEL
LIN {X 0,Y 601.343,Z 481.202,A -85,B 0,C 180,E1 -807.991,E2 -807.991} C_VEL
LIN {X 0,Y 601.339,Z 482.784,A -85,B 0,C 180,E1 -809.33,E2 -809.33} C_VEL
LIN {X 0,Y 601.335,Z 483,A -85,B 0,C 180,E1 -810,E2 -810} C_VEL
LIN {X 0,Y 601.347,Z 482.184,A -85,B 0,C 180,E1 -811.339,E2 -811.339} C_VEL
LIN {X 0,Y 601.343,Z 481.202,A -85,B 0,C 180,E1 -812.009,E2 -812.009} C_VEL
LIN {X 0,Y 601.325,Z 479.809,A -85,B 0,C 180,E1 -812.68,E2 -812.68} C_VEL
LIN {X 0,Y 601.368,Z 476.896,A -85,B 0,C 180,E1 -813.685,E2 -813.685} C_VEL
LIN {X 0,Y 601.336,Z 472.949,A -85,B 0,C 180,E1 -814.693,E2 -814.693} C_VEL
LIN {X 0,Y 601.372,Z 466.877,A -85,B 0,C 180,E1 -815.869,E2 -815.869} C_VEL
LIN {X 0,Y 601.382,Z 460.235,A -85,B 0,C 180,E1 -816.88,E2 -816.88} C_VEL
LIN {X 0,Y 601.401,Z 451.989,A -85,B 0,C 180,E1 -817.892,E2 -817.892} C_VEL
LIN {X 0,Y 601.436,Z 443.536,A -85,B 0,C 180,E1 -818.738,E2 -818.738} C_VEL
LIN {X 0,Y 601.448,Z 433.092,A -85,B 0,C 180,E1 -819.585,E2 -819.585} C_VEL
LIN {X 0,Y 601.478,Z 422.757,A -85,B 0,C 180,E1 -820.264,E2 -820.264} C_VEL
LIN {X 0,Y 601.539,Z 410.582,A -85,B 0,C 180,E1 -820.897,E2 -820.897} C_VEL
LIN {X 0,Y 601.548,Z 398.214,A -85,B 0,C 180,E1 -821.379,E2 -821.379} C_VEL
LIN {X 0,Y 601.568,Z 385.436,A -85,B 0,C 180,E1 -821.733,E2 -821.733} C_VEL
LIN {X 0,Y 601.61,Z 373.082,A -85,B 0,C 180,E1 -821.946,E2 -821.946} C_VEL
LIN {X 0,Y 601.551,Z 271.811,A -85,B 0,C 180,E1 -823.161,E2 -823.161} C_VEL
LIN {X 0,Y 601.457,Z 270.635,A -85,B 0,C 180,E1 -823.214,E2 -823.214} C_VEL
LIN {X 0,Y 601.484,Z 250.8,A -85,B 0,C 180,E1 -825.937,E2 -825.937} C_VEL
LIN {X 0,Y 601.535,Z 231.492,A -85,B 0,C 180,E1 -828.623,E2 -828.623} C_VEL
LIN {X 0,Y 601.636,Z 211.761,A -85,B 0,C 180,E1 -831.41,E2 -831.41} C_VEL
LIN {X 0,Y 601.403,Z 204.617,A -85,B 0,C 180,E1 -832.443,E2 -832.443} C_VEL
LIN {X 0,Y 601.391,Z 204.57,A -85,B 0,C 180,E1 -834.879,E2 -834.879} C_VEL
LIN {X 0,Y 601.397,Z 204.57,A -85,B 0,C 180,E1 -837.868,E2 -837.868} C_VEL
LIN {X 0,Y 601.407,Z 204.566,A -85,B 0,C 180,E1 -840.165,E2 -840.165} C_VEL
LIN {X 0,Y 601.408,Z 204.566,A -85,B 0,C 180,E1 -842.713,E2 -842.713} C_VEL
LIN {X 0,Y 601.385,Z 204.574,A -85,B 0,C 180,E1 -845.11,E2 -845.11} C_VEL
LIN {X 0,Y 601.435,Z 204.571,A -85,B 0,C 180,E1 -847.419,E2 -847.419} C_VEL
LIN {X 0,Y 601.402,Z 204.567,A -85,B 0,C 180,E1 -849.996,E2 -849.996} C_VEL
LIN {X 0,Y 601.406,Z 204.567,A -85,B 0,C 180,E1 -852.671,E2 -852.671} C_VEL
LIN {X 0,Y 601.427,Z 204.569,A -85,B 0,C 180,E1 -855.482,E2 -855.482} C_VEL
LIN {X 0,Y 601.418,Z 204.564,A -85,B 0,C 180,E1 -858.407,E2 -858.407} C_VEL
LIN {X 0,Y 601.433,Z 204.567,A -85,B 0,C 180,E1 -861.529,E2 -861.529} C_VEL
LIN {X 0,Y 601.405,Z 204.565,A -85,B 0,C 180,E1 -864.246,E2 -864.246} C_VEL
LIN {X 0,Y 601.414,Z 204.567,A -85,B 0,C 180,E1 -866.686,E2 -866.686} C_VEL
LIN {X 0,Y 601.415,Z 204.574,A -85,B 0,C 180,E1 -869.058,E2 -869.058} C_VEL
LIN {X 0,Y 601.431,Z 204.568,A -85,B 0,C 180,E1 -871.373,E2 -871.373} C_VEL
LIN {X 0,Y 601.4,Z 204.568,A -85,B 0,C 180,E1 -873.636,E2 -873.636} C_VEL
LIN {X 0,Y 601.418,Z 204.567,A -85,B 0,C 180,E1 -876.59,E2 -876.59} C_VEL
LIN {X 0,Y 601.427,Z 204.566,A -85,B 0,C 180,E1 -879.478,E2 -879.478} C_VEL
LIN {X 0,Y 601.395,Z 204.567,A -85,B 0,C 180,E1 -882.312,E2 -882.312} C_VEL
LIN {X 0,Y 601.414,Z 204.566,A -85,B 0,C 180,E1 -884.409,E2 -884.409} C_VEL
LIN {X 0,Y 601.415,Z 204.571,A -85,B 0,C 180,E1 -887.172,E2 -887.172} C_VEL
LIN {X 0,Y 601.432,Z 204.562,A -85,B 0,C 180,E1 -889.905,E2 -889.905} C_VEL
LIN {X 0,Y 601.455,Z 204.565,A -85,B 0,C 180,E1 -892.615,E2 -892.615} C_VEL
LIN {X 0,Y 601.411,Z 204.568,A -85,B 0,C 180,E1 -895.308,E2 -895.308} C_VEL
LIN {X 0,Y 601.434,Z 204.562,A -85,B 0,C 180,E1 -897.991,E2 -897.991} C_VEL
LIN {X 0,Y 601.454,Z 204.567,A -85,B 0,C 180,E1 -900.67,E2 -900.67} C_VEL
LIN {X 0,Y 601.416,Z 204.566,A -85,B 0,C 180,E1 -903.35,E2 -903.35} C_VEL
LIN {X 0,Y 601.435,Z 204.562,A -85,B 0,C 180,E1 -906.037,E2 -906.037} C_VEL
LIN {X 0,Y 601.434,Z 204.572,A -85,B 0,C 180,E1 -908.738,E2 -908.738} C_VEL
LIN {X 0,Y 601.41,Z 204.565,A -85,B 0,C 180,E1 -911.459,E2 -911.459} C_VEL
LIN {X 0,Y 601.408,Z 204.568,A -85,B 0,C 180,E1 -912.376,E2 -912.376} C_VEL
LIN {X 0,Y 600.74,Z 204.657,A -85,B 0,C 180,E1 -912.935,E2 -912.935} C_VEL
LIN {X 0,Y 597.888,Z 205.012,A -85,B 0,C 180,E1 -913.843,E2 -913.843} C_VEL
LIN {X 0,Y 595.477,Z 205.312,A -85,B 0,C 180,E1 -914.573,E2 -914.573} C_VEL
LIN {X 0,Y 594.439,Z 205.436,A -85,B 0,C 180,E1 -915.137,E2 -915.137} C_VEL
LIN {X 0,Y 594.353,Z 205.445,A -85,B 0,C 180,E1 -915.327,E2 -915.327} C_VEL
LIN {X 0,Y 594.385,Z 205.442,A -85,B 0,C 180,E1 -917.194,E2 -917.194} C_VEL
LIN {X 0,Y 594.371,Z 205.443,A -85,B 0,C 180,E1 -920.054,E2 -920.054} C_VEL
LIN {X 0,Y 594.354,Z 205.448,A -85,B 0,C 180,E1 -922.968,E2 -922.968} C_VEL
LIN {X 0,Y 594.356,Z 205.445,A -85,B 0,C 180,E1 -925.194,E2 -925.194} C_VEL
LIN {X 0,Y 594.341,Z 205.445,A -85,B 0,C 180,E1 -927.519,E2 -927.519} C_VEL
LIN {X 0,Y 594.384,Z 205.447,A -85,B 0,C 180,E1 -930.328,E2 -930.328} C_VEL
LIN {X 0,Y 594.375,Z 205.445,A -85,B 0,C 180,E1 -932.951,E2 -932.951} C_VEL
LIN {X 0,Y 594.325,Z 205.448,A -85,B 0,C 180,E1 -935.411,E2 -935.411} C_VEL
LIN {X 0,Y 594.373,Z 205.444,A -85,B 0,C 180,E1 -937.942,E2 -937.942} C_VEL
LIN {X 0,Y 594.363,Z 205.447,A -85,B 0,C 180,E1 -940.821,E2 -940.821} C_VEL
LIN {X 0,Y 594.349,Z 205.445,A -85,B 0,C 180,E1 -943.301,E2 -943.301} C_VEL
LIN {X 0,Y 594.399,Z 205.613,A -85,B 0,C 180,E1 -945.565,E2 -945.565} C_VEL
LIN {X 0,Y 594.48,Z 217.753,A -85,B 0,C 180,E1 -947.635,E2 -947.635} C_VEL
LIN {X 0,Y 594.373,Z 235.058,A -85,B 0,C 180,E1 -950.539,E2 -950.539} C_VEL
LIN {X 0,Y 594.394,Z 242.145,A -85,B 0,C 180,E1 -951.719,E2 -951.719} C_VEL
LIN {X 0,Y 594.77,Z 246.845,A -85,B 0,C 180,E1 -951.793,E2 -951.793} C_VEL
LIN {X 0,Y 594.621,Z 349.317,A -85,B 0,C 180,E1 -953.05,E2 -953.05} C_VEL
LIN {X 0,Y 594.592,Z 362.924,A -85,B 0,C 180,E1 -953.365,E2 -953.365} C_VEL
LIN {X 0,Y 594.574,Z 374.781,A -85,B 0,C 180,E1 -953.771,E2 -953.771} C_VEL
LIN {X 0,Y 594.516,Z 386.172,A -85,B 0,C 180,E1 -954.29,E2 -954.29} C_VEL
LIN {X 0,Y 594.451,Z 396.809,A -85,B 0,C 180,E1 -954.909,E2 -954.909} C_VEL
LIN {X 0,Y 594.421,Z 407.328,A -85,B 0,C 180,E1 -955.672,E2 -955.672} C_VEL
LIN {X 0,Y 594.364,Z 417.089,A -85,B 0,C 180,E1 -956.543,E2 -956.543} C_VEL
LIN {X 0,Y 594.356,Z 425.378,A -85,B 0,C 180,E1 -957.451,E2 -957.451} C_VEL
LIN {X 0,Y 594.327,Z 432.235,A -85,B 0,C 180,E1 -958.366,E2 -958.366} C_VEL
LIN {X 0,Y 594.289,Z 438.716,A -85,B 0,C 180,E1 -959.435,E2 -959.435} C_VEL
LIN {X 0,Y 594.276,Z 444.252,A -85,B 0,C 180,E1 -960.608,E2 -960.608} C_VEL
LIN {X 0,Y 594.24,Z 448.303,A -85,B 0,C 180,E1 -961.766,E2 -961.766} C_VEL
LIN {X 0,Y 594.265,Z 450.247,A -85,B 0,C 180,E1 -962.534,E2 -962.534} C_VEL
LIN {X 0,Y 594.226,Z 451.659,A -85,B 0,C 180,E1 -963.293,E2 -963.293} C_VEL
LIN {X 0,Y 594.229,Z 452.564,A -85,B 0,C 180,E1 -964.049,E2 -964.049} C_VEL
LIN {X 0,Y 594.22,Z 452.95,A -85,B 0,C 180,E1 -964.8,E2 -964.8} C_VEL
LIN {X 0,Y 594.215,Z 452.864,A -85,B 0,C 180,E1 -965.604,E2 -965.604} C_VEL
LIN {X 0,Y 594.224,Z 452.313,A -85,B 0,C 180,E1 -966.289,E2 -966.289} C_VEL
LIN {X 0,Y 594.247,Z 450.803,A -85,B 0,C 180,E1 -967.293,E2 -967.293} C_VEL
LIN {X 0,Y 594.248,Z 447.778,A -85,B 0,C 180,E1 -968.492,E2 -968.492} C_VEL
LIN {X 0,Y 594.284,Z 443.835,A -85,B 0,C 180,E1 -969.582,E2 -969.582} C_VEL
LIN {X 0,Y 594.298,Z 438.67,A -85,B 0,C 180,E1 -970.663,E2 -970.663} C_VEL
LIN {X 0,Y 594.323,Z 432.146,A -85,B 0,C 180,E1 -971.738,E2 -971.738} C_VEL
LIN {X 0,Y 594.328,Z 423.965,A -85,B 0,C 180,E1 -972.805,E2 -972.805} C_VEL
LIN {X 0,Y 594.403,Z 415.586,A -85,B 0,C 180,E1 -973.691,E2 -973.691} C_VEL
LIN {X 0,Y 594.449,Z 405.394,A -85,B 0,C 180,E1 -974.573,E2 -974.573} C_VEL
LIN {X 0,Y 594.453,Z 395.34,A -85,B 0,C 180,E1 -975.275,E2 -975.275} C_VEL
LIN {X 0,Y 594.533,Z 384.004,A -85,B 0,C 180,E1 -975.907,E2 -975.907} C_VEL
LIN {X 0,Y 594.586,Z 371.188,A -85,B 0,C 180,E1 -976.456,E2 -976.456} C_VEL
LIN {X 0,Y 594.575,Z 358.414,A -85,B 0,C 180,E1 -976.848,E2 -976.848} C_VEL
LIN {X 0,Y 594.609,Z 344.807,A -85,B 0,C 180,E1 -977.109,E2 -977.109} C_VEL
LIN {X 0,Y 594.683,Z 243.967,A -85,B 0,C 180,E1 -978.334,E2 -978.334} C_VEL
LIN {X 0,Y 594.378,Z 242.078,A -85,B 0,C 180,E1 -978.382,E2 -978.382} C_VEL
LIN {X 0,Y 594.391,Z 228.524,A -85,B 0,C 180,E1 -980.643,E2 -980.643} C_VEL
LIN {X 0,Y 594.475,Z 213.302,A -85,B 0,C 180,E1 -983.21,E2 -983.21} C_VEL
LIN {X 0,Y 594.363,Z 205.446,A -85,B 0,C 180,E1 -984.572,E2 -984.572} C_VEL
LIN {X 0,Y 594.385,Z 205.445,A -85,B 0,C 180,E1 -987.289,E2 -987.289} C_VEL
LIN {X 0,Y 594.414,Z 205.441,A -85,B 0,C 180,E1 -990,E2 -990} C_VEL
LIN {X 0,Y 594.374,Z 205.441,A -85,B 0,C 180,E1 -992.711,E2 -992.711} C_VEL
LIN {X 0,Y 594.376,Z 205.448,A -85,B 0,C 180,E1 -995.428,E2 -995.428} C_VEL
LIN {X 0,Y 594.381,Z 205.442,A -85,B 0,C 180,E1 -998.157,E2 -998.157} C_VEL
LIN {X 0,Y 594.371,Z 205.444,A -85,B 0,C 180,E1 -1001.062,E2 -1001.062} C_VEL
LIN {X 0,Y 594.376,Z 205.45,A -85,B 0,C 180,E1 -1003.679,E2 -1003.679} C_VEL
LIN {X 0,Y 594.345,Z 205.445,A -85,B 0,C 180,E1 -1006.702,E2 -1006.702} C_VEL
LIN {X 0,Y 594.363,Z 205.45,A -85,B 0,C 180,E1 -1009.334,E2 -1009.334} C_VEL
LIN {X 0,Y 594.359,Z 205.454,A -85,B 0,C 180,E1 -1011.503,E2 -1011.503} C_VEL
LIN {X 0,Y 594.369,Z 205.442,A -85,B 0,C 180,E1 -1014.447,E2 -1014.447} C_VEL
LIN {X 0,Y 594.364,Z 205.443,A -85,B 0,C 180,E1 -1016.7,E2 -1016.7} C_VEL
LIN {X 0,Y 594.374,Z 205.445,A -85,B 0,C 180,E1 -1018.999,E2 -1018.999} C_VEL
LIN {X 0,Y 594.375,Z 205.448,A -85,B 0,C 180,E1 -1021.642,E2 -1021.642} C_VEL
LIN {X 0,Y 594.369,Z 205.442,A -85,B 0,C 180,E1 -1024.58,E2 -1024.58} C_VEL
LIN {X 0,Y 594.387,Z 205.446,A -85,B 0,C 180,E1 -1027.608,E2 -1027.608} C_VEL
LIN {X 0,Y 594.363,Z 205.443,A -85,B 0,C 180,E1 -1030.567,E2 -1030.567} C_VEL
LIN {X 0,Y 594.36,Z 205.453,A -85,B 0,C 180,E1 -1033.3,E2 -1033.3} C_VEL
LIN {X 0,Y 594.366,Z 205.443,A -85,B 0,C 180,E1 -1036.16,E2 -1036.16} C_VEL
LIN {X 0,Y 594.373,Z 205.442,A -85,B 0,C 180,E1 -1038.535,E2 -1038.535} C_VEL
LIN {X 0,Y 594.379,Z 205.451,A -85,B 0,C 180,E1 -1041.296,E2 -1041.296} C_VEL
LIN {X 0,Y 594.393,Z 205.442,A -85,B 0,C 180,E1 -1043.758,E2 -1043.758} C_VEL
LIN {X 0,Y 594.374,Z 205.441,A -85,B 0,C 180,E1 -1046.238,E2 -1046.238} C_VEL
LIN {X 0,Y 594.366,Z 205.444,A -85,B 0,C 180,E1 -1048.649,E2 -1048.649} C_VEL
LIN {X 0,Y 594.382,Z 205.448,A -85,B 0,C 180,E1 -1051.042,E2 -1051.042} C_VEL
LIN {X 0,Y 594.38,Z 205.441,A -85,B 0,C 180,E1 -1053.978,E2 -1053.978} C_VEL
LIN {X 0,Y 594.39,Z 205.44,A -85,B 0,C 180,E1 -1056.296,E2 -1056.296} C_VEL
LIN {X 0,Y 594.404,Z 205.447,A -85,B 0,C 180,E1 -1059.224,E2 -1059.224} C_VEL
LIN {X 0,Y 594.352,Z 205.444,A -85,B 0,C 180,E1 -1062.095,E2 -1062.095} C_VEL
LIN {X 0,Y 594.363,Z 205.443,A -85,B 0,C 180,E1 -1064.219,E2 -1064.219} C_VEL
LIN {X 0,Y 594.379,Z 205.441,A -85,B 0,C 180,E1 -1066.321,E2 -1066.321} C_VEL
LIN {X 0,Y 594.376,Z 205.451,A -85,B 0,C 180,E1 -1069.095,E2 -1069.095} C_VEL
LIN {X 0,Y 594.415,Z 205.437,A -85,B 0,C 180,E1 -1071.843,E2 -1071.843} C_VEL
LIN {X 0,Y 594.393,Z 205.442,A -85,B 0,C 180,E1 -1074.572,E2 -1074.572} C_VEL
LIN {X 0,Y 594.403,Z 205.444,A -85,B 0,C 180,E1 -1077.289,E2 -1077.289} C_VEL
LIN {X 0,Y 594.413,Z 205.436,A -85,B 0,C 180,E1 -1080,E2 -1080} C_VEL
LIN {X 0,Y 594.402,Z 205.444,A -85,B 0,C 180,E1 -1082.711,E2 -1082.711} C_VEL
LIN {X 0,Y 594.394,Z 205.442,A -85,B 0,C 180,E1 -1085.428,E2 -1085.428} C_VEL
LIN {X 0,Y 594.412,Z 205.437,A -85,B 0,C 180,E1 -1088.157,E2 -1088.157} C_VEL
LIN {X 0,Y 594.388,Z 205.448,A -85,B 0,C 180,E1 -1091.075,E2 -1091.075} C_VEL
LIN {X 0,Y 594.379,Z 205.441,A -85,B 0,C 180,E1 -1093.679,E2 -1093.679} C_VEL
LIN {X 0,Y 594.391,Z 205.447,A -85,B 0,C 180,E1 -1096.72,E2 -1096.72} C_VEL
LIN {X 0,Y 594.364,Z 205.446,A -85,B 0,C 180,E1 -1099.335,E2 -1099.335} C_VEL
LIN {X 0,Y 594.363,Z 205.444,A -85,B 0,C 180,E1 -1101.503,E2 -1101.503} C_VEL
LIN {X 0,Y 594.387,Z 205.444,A -85,B 0,C 180,E1 -1104.446,E2 -1104.446} C_VEL
LIN {X 0,Y 594.379,Z 205.449,A -85,B 0,C 180,E1 -1106.7,E2 -1106.7} C_VEL
LIN {X 0,Y 594.379,Z 205.448,A -85,B 0,C 180,E1 -1108.999,E2 -1108.999} C_VEL
LIN {X 0,Y 594.374,Z 205.441,A -85,B 0,C 180,E1 -1111.643,E2 -1111.643} C_VEL
LIN {X 0,Y 594.384,Z 205.447,A -85,B 0,C 180,E1 -1114.58,E2 -1114.58} C_VEL
LIN {X 0,Y 594.381,Z 205.445,A -85,B 0,C 180,E1 -1117.087,E2 -1117.087} C_VEL
LIN {X 0,Y 594.354,Z 205.444,A -85,B 0,C 180,E1 -1119.772,E2 -1119.772} C_VEL
LIN {X 0,Y 594.367,Z 205.447,A -85,B 0,C 180,E1 -1122.376,E2 -1122.376} C_VEL
LIN {X 0,Y 594.343,Z 205.448,A -85,B 0,C 180,E1 -1125.194,E2 -1125.194} C_VEL
LIN {X 0,Y 594.363,Z 205.443,A -85,B 0,C 180,E1 -1127.625,E2 -1127.625} C_VEL
LIN {X 0,Y 594.373,Z 205.446,A -85,B 0,C 180,E1 -1130.32,E2 -1130.32} C_VEL
LIN {X 0,Y 594.378,Z 205.446,A -85,B 0,C 180,E1 -1132.913,E2 -1132.913} C_VEL
LIN {X 0,Y 594.376,Z 205.442,A -85,B 0,C 180,E1 -1135.863,E2 -1135.863} C_VEL
LIN {X 0,Y 594.366,Z 205.452,A -85,B 0,C 180,E1 -1138.65,E2 -1138.65} C_VEL
LIN {X 0,Y 594.375,Z 205.444,A -85,B 0,C 180,E1 -1141.044,E2 -1141.044} C_VEL
LIN {X 0,Y 594.364,Z 205.444,A -85,B 0,C 180,E1 -1143.3,E2 -1143.3} C_VEL
LIN {X 0,Y 594.376,Z 205.442,A -85,B 0,C 180,E1 -1145.57,E2 -1145.57} C_VEL
LIN {X 0,Y 594.378,Z 205.553,A -85,B 0,C 180,E1 -1147.414,E2 -1147.414} C_VEL
LIN {X 0,Y 594.745,Z 209.244,A -85,B 0,C 180,E1 -1147.965,E2 -1147.965} C_VEL
LIN {X 0,Y 594.628,Z 229.721,A -85,B 0,C 180,E1 -1150.9,E2 -1150.9} C_VEL
LIN {X 0,Y 594.5,Z 249.543,A -85,B 0,C 180,E1 -1153.694,E2 -1153.694} C_VEL
LIN {X 0,Y 594.423,Z 269.692,A -85,B 0,C 180,E1 -1156.496,E2 -1156.496} C_VEL
LIN {X 0,Y 594.46,Z 271.158,A -85,B 0,C 180,E1 -1156.671,E2 -1156.671} C_VEL
LIN {X 0,Y 594.74,Z 280.102,A -85,B 0,C 180,E1 -1156.787,E2 -1156.787} C_VEL
LIN {X 0,Y 594.654,Z 378.957,A -85,B 0,C 180,E1 -1157.999,E2 -1157.999} C_VEL
LIN {X 0,Y 594.626,Z 392.225,A -85,B 0,C 180,E1 -1158.301,E2 -1158.301} C_VEL
LIN {X 0,Y 594.567,Z 404.622,A -85,B 0,C 180,E1 -1158.72,E2 -1158.72} C_VEL
LIN {X 0,Y 594.533,Z 416.635,A -85,B 0,C 180,E1 -1159.27,E2 -1159.27} C_VEL
LIN {X 0,Y 594.472,Z 428.203,A -85,B 0,C 180,E1 -1159.958,E2 -1159.958} C_VEL
LIN {X 0,Y 594.414,Z 438.599,A -85,B 0,C 180,E1 -1160.73,E2 -1160.73} C_VEL
LIN {X 0,Y 594.383,Z 447.114,A -85,B 0,C 180,E1 -1161.501,E2 -1161.501} C_VEL
LIN {X 0,Y 594.347,Z 454.962,A -85,B 0,C 180,E1 -1162.356,E2 -1162.356} C_VEL
LIN {X 0,Y 594.282,Z 462.813,A -85,B 0,C 180,E1 -1163.408,E2 -1163.408} C_VEL
LIN {X 0,Y 594.289,Z 469.681,A -85,B 0,C 180,E1 -1164.571,E2 -1164.571} C_VEL
LIN {X 0,Y 594.27,Z 474.372,A -85,B 0,C 180,E1 -1165.591,E2 -1165.591} C_VEL
LIN {X 0,Y 594.267,Z 477.957,A -85,B 0,C 180,E1 -1166.61,E2 -1166.61} C_VEL
LIN {X 0,Y 594.226,Z 479.809,A -85,B 0,C 180,E1 -1167.289,E2 -1167.289} C_VEL
LIN {X 0,Y 594.241,Z 481.201,A -85,B 0,C 180,E1 -1167.967,E2 -1167.967} C_VEL
LIN {X 0,Y 594.239,Z 482.784,A -85,B 0,C 180,E1 -1169.322,E2 -1169.322} C_VEL
LIN {X 0,Y 594.236,Z 483,A -85,B 0,C 180,E1 -1170,E2 -1170} C_VEL
LIN {X 0,Y 594.247,Z 482.185,A -85,B 0,C 180,E1 -1171.355,E2 -1171.355} C_VEL
LIN {X 0,Y 594.241,Z 481.201,A -85,B 0,C 180,E1 -1172.033,E2 -1172.033} C_VEL
LIN {X 0,Y 594.226,Z 479.809,A -85,B 0,C 180,E1 -1172.712,E2 -1172.712} C_VEL
LIN {X 0,Y 594.289,Z 476.896,A -85,B 0,C 180,E1 -1173.729,E2 -1173.729} C_VEL
LIN {X 0,Y 594.241,Z 472.949,A -85,B 0,C 180,E1 -1174.749,E2 -1174.749} C_VEL
LIN {X 0,Y 594.304,Z 466.877,A -85,B 0,C 180,E1 -1175.939,E2 -1175.939} C_VEL
LIN {X 0,Y 594.308,Z 460.236,A -85,B 0,C 180,E1 -1176.962,E2 -1176.962} C_VEL
LIN {X 0,Y 594.359,Z 451.989,A -85,B 0,C 180,E1 -1177.986,E2 -1177.986} C_VEL
LIN {X 0,Y 594.382,Z 443.537,A -85,B 0,C 180,E1 -1178.842,E2 -1178.842} C_VEL
LIN {X 0,Y 594.431,Z 433.094,A -85,B 0,C 180,E1 -1179.699,E2 -1179.699} C_VEL
LIN {X 0,Y 594.489,Z 422.758,A -85,B 0,C 180,E1 -1180.386,E2 -1180.386} C_VEL
LIN {X 0,Y 594.559,Z 411.71,A -85,B 0,C 180,E1 -1180.974,E2 -1180.974} C_VEL
LIN {X 0,Y 594.573,Z 399.706,A -85,B 0,C 180,E1 -1181.464,E2 -1181.464} C_VEL
LIN {X 0,Y 594.607,Z 386.349,A -85,B 0,C 180,E1 -1181.851,E2 -1181.851} C_VEL
LIN {X 0,Y 594.662,Z 373.082,A -85,B 0,C 180,E1 -1182.088,E2 -1182.088} C_VEL
LIN {X 0,Y 594.702,Z 272.929,A -85,B 0,C 180,E1 -1183.302,E2 -1183.302} C_VEL
LIN {X 0,Y 594.422,Z 270.792,A -85,B 0,C 180,E1 -1183.351,E2 -1183.351} C_VEL
LIN {X 0,Y 594.502,Z 250.8,A -85,B 0,C 180,E1 -1186.129,E2 -1186.129} C_VEL
LIN {X 0,Y 594.6,Z 231.303,A -85,B 0,C 180,E1 -1188.875,E2 -1188.875} C_VEL
LIN {X 0,Y 594.751,Z 211.761,A -85,B 0,C 180,E1 -1191.671,E2 -1191.671} C_VEL
LIN {X 0,Y 594.463,Z 206.028,A -85,B 0,C 180,E1 -1192.514,E2 -1192.514} C_VEL
LIN {X 0,Y 594.378,Z 205.446,A -85,B 0,C 180,E1 -1192.621,E2 -1192.621} C_VEL
LIN {X 0,Y 594.371,Z 205.449,A -85,B 0,C 180,E1 -1195.193,E2 -1195.193} C_VEL
LIN {X 0,Y 594.37,Z 205.451,A -85,B 0,C 180,E1 -1197.523,E2 -1197.523} C_VEL
LIN {X 0,Y 594.371,Z 205.442,A -85,B 0,C 180,E1 -1200.325,E2 -1200.325} C_VEL
LIN {X 0,Y 594.377,Z 205.445,A -85,B 0,C 180,E1 -1202.95,E2 -1202.95} C_VEL
LIN {X 0,Y 594.348,Z 205.454,A -85,B 0,C 180,E1 -1205.409,E2 -1205.409} C_VEL
LIN {X 0,Y 594.383,Z 205.442,A -85,B 0,C 180,E1 -1207.941,E2 -1207.941} C_VEL
LIN {X 0,Y 594.373,Z 205.444,A -85,B 0,C 180,E1 -1210.821,E2 -1210.821} C_VEL
LIN {X 0,Y 594.376,Z 205.443,A -85,B 0,C 180,E1 -1213.84,E2 -1213.84} C_VEL
LIN {X 0,Y 594.365,Z 205.445,A -85,B 0,C 180,E1 -1216.7,E2 -1216.7} C_VEL
LIN {X 0,Y 594.371,Z 205.448,A -85,B 0,C 180,E1 -1219.433,E2 -1219.433} C_VEL
LIN {X 0,Y 594.388,Z 205.44,A -85,B 0,C 180,E1 -1222.391,E2 -1222.391} C_VEL
LIN {X 0,Y 594.357,Z 205.446,A -85,B 0,C 180,E1 -1224.675,E2 -1224.675} C_VEL
LIN {X 0,Y 594.376,Z 205.451,A -85,B 0,C 180,E1 -1227.089,E2 -1227.089} C_VEL
LIN {X 0,Y 594.386,Z 205.442,A -85,B 0,C 180,E1 -1229.672,E2 -1229.672} C_VEL
LIN {X 0,Y 594.374,Z 205.443,A -85,B 0,C 180,E1 -1232.539,E2 -1232.539} C_VEL
LIN {X 0,Y 594.373,Z 205.447,A -85,B 0,C 180,E1 -1234.807,E2 -1234.807} C_VEL
LIN {X 0,Y 594.364,Z 205.449,A -85,B 0,C 180,E1 -1237.265,E2 -1237.265} C_VEL
LIN {X 0,Y 594.372,Z 205.441,A -85,B 0,C 180,E1 -1239.946,E2 -1239.946} C_VEL
LIN {X 0,Y 594.382,Z 205.447,A -85,B 0,C 180,E1 -1242.806,E2 -1242.806} C_VEL
LIN {X 0,Y 594.388,Z 205.439,A -85,B 0,C 180,E1 -1245.826,E2 -1245.826} C_VEL
LIN {X 0,Y 594.395,Z 205.441,A -85,B 0,C 180,E1 -1248.404,E2 -1248.404} C_VEL
LIN {X 0,Y 594.377,Z 205.447,A -85,B 0,C 180,E1 -1251.158,E2 -1251.158} C_VEL
LIN {X 0,Y 594.383,Z 205.44,A -85,B 0,C 180,E1 -1253.891,E2 -1253.891} C_VEL
LIN {X 0,Y 594.386,Z 205.446,A -85,B 0,C 180,E1 -1256.611,E2 -1256.611} C_VEL
LIN {X 0,Y 594.41,Z 205.439,A -85,B 0,C 180,E1 -1259.323,E2 -1259.323} C_VEL
LIN {X 0,Y 594.404,Z 205.438,A -85,B 0,C 180,E1 -1262.033,E2 -1262.033} C_VEL
LIN {X 0,Y 594.392,Z 205.449,A -85,B 0,C 180,E1 -1264.748,E2 -1264.748} C_VEL
LIN {X 0,Y 594.369,Z 205.442,A -85,B 0,C 180,E1 -1267.474,E2 -1267.474} C_VEL
LIN {X 0,Y 594.392,Z 205.441,A -85,B 0,C 180,E1 -1270.216,E2 -1270.216} C_VEL
LIN {X 0,Y 594.362,Z 205.448,A -85,B 0,C 180,E1 -1272.983,E2 -1272.983} C_VEL
LIN {X 0,Y 594.353,Z 205.445,A -85,B 0,C 180,E1 -1275.327,E2 -1275.327} C_VEL
LIN {X 0,Y 593.679,Z 205.529,A -85,B 0,C 180,E1 -1275.893,E2 -1275.893} C_VEL
LIN {X 0,Y 590.815,Z 205.893,A -85,B 0,C 180,E1 -1276.811,E2 -1276.811} C_VEL
LIN {X 0,Y 588.407,Z 206.19,A -85,B 0,C 180,E1 -1277.55,E2 -1277.55} C_VEL
LIN {X 0,Y 587.385,Z 206.314,A -85,B 0,C 180,E1 -1278.12,E2 -1278.12} C_VEL
LIN {X 0,Y 587.308,Z 206.324,A -85,B 0,C 180,E1 -1278.313,E2 -1278.313} C_VEL
LIN {X 0,Y 587.33,Z 206.322,A -85,B 0,C 180,E1 -1281.038,E2 -1281.038} C_VEL
LIN {X 0,Y 587.313,Z 206.322,A -85,B 0,C 180,E1 -1283.259,E2 -1283.259} C_VEL
LIN {X 0,Y 587.32,Z 206.32,A -85,B 0,C 180,E1 -1285.518,E2 -1285.518} C_VEL
LIN {X 0,Y 587.304,Z 206.323,A -85,B 0,C 180,E1 -1287.82,E2 -1287.82} C_VEL
LIN {X 0,Y 587.333,Z 206.328,A -85,B 0,C 180,E1 -1290.51,E2 -1290.51} C_VEL
LIN {X 0,Y 587.326,Z 206.32,A -85,B 0,C 180,E1 -1293.397,E2 -1293.397} C_VEL
LIN {X 0,Y 587.281,Z 206.327,A -85,B 0,C 180,E1 -1295.901,E2 -1295.901} C_VEL
LIN {X 0,Y 587.316,Z 206.331,A -85,B 0,C 180,E1 -1298.481,E2 -1298.481} C_VEL
LIN {X 0,Y 587.31,Z 206.323,A -85,B 0,C 180,E1 -1301.159,E2 -1301.159} C_VEL
LIN {X 0,Y 587.303,Z 206.328,A -85,B 0,C 180,E1 -1304.111,E2 -1304.111} C_VEL
LIN {X 0,Y 587.339,Z 206.38,A -85,B 0,C 180,E1 -1305.454,E2 -1305.454} C_VEL
LIN {X 0,Y 587.512,Z 212.418,A -85,B 0,C 180,E1 -1306.504,E2 -1306.504} C_VEL
LIN {X 0,Y 587.394,Z 229.011,A -85,B 0,C 180,E1 -1309.339,E2 -1309.339} C_VEL
LIN {X 0,Y 587.359,Z 242.249,A -85,B 0,C 180,E1 -1311.566,E2 -1311.566} C_VEL
LIN {X 0,Y 587.86,Z 246.935,A -85,B 0,C 180,E1 -1311.635,E2 -1311.635} C_VEL
LIN {X 0,Y 587.689,Z 349.167,A -85,B 0,C 180,E1 -1312.904,E2 -1312.904} C_VEL
LIN {X 0,Y 587.663,Z 362.175,A -85,B 0,C 180,E1 -1313.204,E2 -1313.204} C_VEL
LIN {X 0,Y 587.606,Z 375.02,A -85,B 0,C 180,E1 -1313.645,E2 -1313.645} C_VEL
LIN {X 0,Y 587.506,Z 387.145,A -85,B 0,C 180,E1 -1314.213,E2 -1314.213} C_VEL
LIN {X 0,Y 587.412,Z 399.227,A -85,B 0,C 180,E1 -1314.95,E2 -1314.95} C_VEL
LIN {X 0,Y 587.379,Z 410.01,A -85,B 0,C 180,E1 -1315.781,E2 -1315.781} C_VEL
LIN {X 0,Y 587.307,Z 418.656,A -85,B 0,C 180,E1 -1316.602,E2 -1316.602} C_VEL
LIN {X 0,Y 587.279,Z 427.432,A -85,B 0,C 180,E1 -1317.621,E2 -1317.621} C_VEL
LIN {X 0,Y 587.242,Z 434.457,A -85,B 0,C 180,E1 -1318.628,E2 -1318.628} C_VEL
LIN {X 0,Y 587.188,Z 441.022,A -85,B 0,C 180,E1 -1319.822,E2 -1319.822} C_VEL
LIN {X 0,Y 587.172,Z 445.576,A -85,B 0,C 180,E1 -1320.898,E2 -1320.898} C_VEL
LIN {X 0,Y 587.159,Z 449.483,A -85,B 0,C 180,E1 -1322.173,E2 -1322.173} C_VEL
LIN {X 0,Y 587.132,Z 451.13,A -85,B 0,C 180,E1 -1322.944,E2 -1322.944} C_VEL
LIN {X 0,Y 587.12,Z 452.406,A -85,B 0,C 180,E1 -1323.867,E2 -1323.867} C_VEL
LIN {X 0,Y 587.118,Z 452.861,A -85,B 0,C 180,E1 -1324.473,E2 -1324.473} C_VEL
LIN {X 0,Y 587.119,Z 452.909,A -85,B 0,C 180,E1 -1325.471,E2 -1325.471} C_VEL
LIN {X 0,Y 587.116,Z 451.796,A -85,B 0,C 180,E1 -1326.733,E2 -1326.733} C_VEL
LIN {X 0,Y 587.148,Z 450.473,A -85,B 0,C 180,E1 -1327.478,E2 -1327.478} C_VEL
LIN {X 0,Y 587.157,Z 447.612,A -85,B 0,C 180,E1 -1328.588,E2 -1328.588} C_VEL
LIN {X 0,Y 587.203,Z 443.613,A -85,B 0,C 180,E1 -1329.691,E2 -1329.691} C_VEL
LIN {X 0,Y 587.23,Z 438.578,A -85,B 0,C 180,E1 -1330.749,E2 -1330.749} C_VEL
LIN {X 0,Y 587.226,Z 431.808,A -85,B 0,C 180,E1 -1331.87,E2 -1331.87} C_VEL
LIN {X 0,Y 587.27,Z 423.574,A -85,B 0,C 180,E1 -1332.944,E2 -1332.944} C_VEL
LIN {X 0,Y 587.353,Z 415.06,A -85,B 0,C 180,E1 -1333.847,E2 -1333.847} C_VEL
LIN {X 0,Y 587.393,Z 404.742,A -85,B 0,C 180,E1 -1334.739,E2 -1334.739} C_VEL
LIN {X 0,Y 587.46,Z 393.503,A -85,B 0,C 180,E1 -1335.511,E2 -1335.511} C_VEL
LIN {X 0,Y 587.582,Z 381.528,A -85,B 0,C 180,E1 -1336.16,E2 -1336.16} C_VEL
LIN {X 0,Y 587.6,Z 369.789,A -85,B 0,C 180,E1 -1336.645,E2 -1336.645} C_VEL
LIN {X 0,Y 587.651,Z 357.122,A -85,B 0,C 180,E1 -1337.02,E2 -1337.02} C_VEL
LIN {X 0,Y 587.676,Z 344.237,A -85,B 0,C 180,E1 -1337.262,E2 -1337.262} C_VEL
LIN {X 0,Y 587.748,Z 244.707,A -85,B 0,C 180,E1 -1338.485,E2 -1338.485} C_VEL
LIN {X 0,Y 587.33,Z 242.065,A -85,B 0,C 180,E1 -1338.548,E2 -1338.548} C_VEL
LIN {X 0,Y 587.415,Z 227.237,A -85,B 0,C 180,E1 -1341.052,E2 -1341.052} C_VEL
LIN {X 0,Y 587.51,Z 211.064,A -85,B 0,C 180,E1 -1343.819,E2 -1343.819} C_VEL
LIN {X 0,Y 587.314,Z 206.325,A -85,B 0,C 180,E1 -1344.679,E2 -1344.679} C_VEL
LIN {X 0,Y 587.37,Z 206.32,A -85,B 0,C 180,E1 -1347.943,E2 -1347.943} C_VEL
LIN {X 0,Y 587.383,Z 206.317,A -85,B 0,C 180,E1 -1350,E2 -1350} C_VEL
LIN {X 0,Y 587.343,Z 206.317,A -85,B 0,C 180,E1 -1352.743,E2 -1352.743} C_VEL
LIN {X 0,Y 587.343,Z 206.325,A -85,B 0,C 180,E1 -1355.493,E2 -1355.493} C_VEL
LIN {X 0,Y 587.34,Z 206.319,A -85,B 0,C 180,E1 -1358.255,E2 -1358.255} C_VEL
LIN {X 0,Y 587.334,Z 206.321,A -85,B 0,C 180,E1 -1361.124,E2 -1361.124} C_VEL
LIN {X 0,Y 587.343,Z 206.318,A -85,B 0,C 180,E1 -1364.25,E2 -1364.25} C_VEL
LIN {X 0,Y 587.309,Z 206.33,A -85,B 0,C 180,E1 -1367.407,E2 -1367.407} C_VEL
LIN {X 0,Y 587.309,Z 206.331,A -85,B 0,C 180,E1 -1369.576,E2 -1369.576} C_VEL
LIN {X 0,Y 587.314,Z 206.327,A -85,B 0,C 180,E1 -1371.774,E2 -1371.774} C_VEL
LIN {X 0,Y 587.315,Z 206.322,A -85,B 0,C 180,E1 -1374.76,E2 -1374.76} C_VEL
LIN {X 0,Y 587.338,Z 206.322,A -85,B 0,C 180,E1 -1377.818,E2 -1377.818} C_VEL
LIN {X 0,Y 587.322,Z 206.32,A -85,B 0,C 180,E1 -1380.507,E2 -1380.507} C_VEL
LIN {X 0,Y 587.335,Z 206.328,A -85,B 0,C 180,E1 -1383.396,E2 -1383.396} C_VEL
LIN {X 0,Y 587.289,Z 206.327,A -85,B 0,C 180,E1 -1385.9,E2 -1385.9} C_VEL
LIN {X 0,Y 587.32,Z 206.32,A -85,B 0,C 180,E1 -1388.48,E2 -1388.48} C_VEL
LIN {X 0,Y 587.335,Z 206.325,A -85,B 0,C 180,E1 -1391.157,E2 -1391.157} C_VEL
LIN {X 0,Y 587.312,Z 206.322,A -85,B 0,C 180,E1 -1394.111,E2 -1394.111} C_VEL
LIN {X 0,Y 587.312,Z 206.326,A -85,B 0,C 180,E1 -1396.993,E2 -1396.993} C_VEL
LIN {X 0,Y 587.312,Z 206.325,A -85,B 0,C 180,E1 -1399.745,E2 -1399.745} C_VEL
LIN {X 0,Y 587.341,Z 206.318,A -85,B 0,C 180,E1 -1402.392,E2 -1402.392} C_VEL
LIN {X 0,Y 587.327,Z 206.324,A -85,B 0,C 180,E1 -1404.944,E2 -1404.944} C_VEL
LIN {X 0,Y 587.336,Z 206.326,A -85,B 0,C 180,E1 -1407.421,E2 -1407.421} C_VEL
LIN {X 0,Y 587.331,Z 206.321,A -85,B 0,C 180,E1 -1409.83,E2 -1409.83} C_VEL
LIN {X 0,Y 587.349,Z 206.317,A -85,B 0,C 180,E1 -1412.307,E2 -1412.307} C_VEL
LIN {X 0,Y 587.348,Z 206.327,A -85,B 0,C 180,E1 -1415.241,E2 -1415.241} C_VEL
LIN {X 0,Y 587.319,Z 206.32,A -85,B 0,C 180,E1 -1418.225,E2 -1418.225} C_VEL
LIN {X 0,Y 587.347,Z 206.327,A -85,B 0,C 180,E1 -1421.151,E2 -1421.151} C_VEL
LIN {X 0,Y 587.321,Z 206.32,A -85,B 0,C 180,E1 -1424.025,E2 -1424.025} C_VEL
LIN {X 0,Y 587.357,Z 206.316,A -85,B 0,C 180,E1 -1426.154,E2 -1426.154} C_VEL
LIN {X 0,Y 587.341,Z 206.326,A -85,B 0,C 180,E1 -1428.962,E2 -1428.962} C_VEL
LIN {X 0,Y 587.368,Z 206.316,A -85,B 0,C 180,E1 -1431.745,E2 -1431.745} C_VEL
LIN {X 0,Y 587.36,Z 206.318,A -85,B 0,C 180,E1 -1434.507,E2 -1434.507} C_VEL
LIN {X 0,Y 587.369,Z 206.321,A -85,B 0,C 180,E1 -1437.257,E2 -1437.257} C_VEL
LIN {X 0,Y 587.382,Z 206.313,A -85,B 0,C 180,E1 -1440,E2 -1440} C_VEL
LIN {X 0,Y 587.369,Z 206.32,A -85,B 0,C 180,E1 -1442.743,E2 -1442.743} C_VEL
LIN {X 0,Y 587.361,Z 206.318,A -85,B 0,C 180,E1 -1445.493,E2 -1445.493} C_VEL
LIN {X 0,Y 587.363,Z 206.316,A -85,B 0,C 180,E1 -1448.255,E2 -1448.255} C_VEL
LIN {X 0,Y 587.345,Z 206.324,A -85,B 0,C 180,E1 -1451.134,E2 -1451.134} C_VEL
LIN {X 0,Y 587.362,Z 206.316,A -85,B 0,C 180,E1 -1454.261,E2 -1454.261} C_VEL
LIN {X 0,Y 587.348,Z 206.319,A -85,B 0,C 180,E1 -1457.406,E2 -1457.406} C_VEL
LIN {X 0,Y 587.328,Z 206.321,A -85,B 0,C 180,E1 -1460.305,E2 -1460.305} C_VEL
LIN {X 0,Y 587.321,Z 206.324,A -85,B 0,C 180,E1 -1463.259,E2 -1463.259} C_VEL
LIN {X 0,Y 587.328,Z 206.32,A -85,B 0,C 180,E1 -1465.517,E2 -1465.517} C_VEL
LIN {X 0,Y 587.345,Z 206.317,A -85,B 0,C 180,E1 -1467.818,E2 -1467.818} C_VEL
LIN {X 0,Y 587.335,Z 206.324,A -85,B 0,C 180,E1 -1470.51,E2 -1470.51} C_VEL
LIN {X 0,Y 587.331,Z 206.32,A -85,B 0,C 180,E1 -1473.397,E2 -1473.397} C_VEL
LIN {X 0,Y 587.317,Z 206.321,A -85,B 0,C 180,E1 -1475.898,E2 -1475.898} C_VEL
LIN {X 0,Y 587.327,Z 206.325,A -85,B 0,C 180,E1 -1478.48,E2 -1478.48} C_VEL
LIN {X 0,Y 587.332,Z 206.322,A -85,B 0,C 180,E1 -1481.157,E2 -1481.157} C_VEL
LIN {X 0,Y 587.325,Z 206.321,A -85,B 0,C 180,E1 -1484.114,E2 -1484.114} C_VEL
LIN {X 0,Y 587.316,Z 206.326,A -85,B 0,C 180,E1 -1486.994,E2 -1486.994} C_VEL
LIN {X 0,Y 587.31,Z 206.321,A -85,B 0,C 180,E1 -1489.746,E2 -1489.746} C_VEL
LIN {X 0,Y 587.342,Z 206.323,A -85,B 0,C 180,E1 -1492.393,E2 -1492.393} C_VEL
LIN {X 0,Y 587.355,Z 206.316,A -85,B 0,C 180,E1 -1495.78,E2 -1495.78} C_VEL
LIN {X 0,Y 587.336,Z 206.322,A -85,B 0,C 180,E1 -1498.231,E2 -1498.231} C_VEL
LIN {X 0,Y 587.345,Z 206.323,A -85,B 0,C 180,E1 -1500.868,E2 -1500.868} C_VEL
LIN {X 0,Y 587.308,Z 206.323,A -85,B 0,C 180,E1 -1503.72,E2 -1503.72} C_VEL
LIN {X 0,Y 587.314,Z 206.325,A -85,B 0,C 180,E1 -1505.993,E2 -1505.993} C_VEL
LIN {X 0,Y 587.331,Z 206.464,A -85,B 0,C 180,E1 -1507.262,E2 -1507.262} C_VEL
LIN {X 0,Y 587.834,Z 210.504,A -85,B 0,C 180,E1 -1507.877,E2 -1507.877} C_VEL
LIN {X 0,Y 587.663,Z 230.068,A -85,B 0,C 180,E1 -1510.715,E2 -1510.715} C_VEL
LIN {X 0,Y 587.52,Z 249.543,A -85,B 0,C 180,E1 -1513.495,E2 -1513.495} C_VEL
LIN {X 0,Y 587.427,Z 269.692,A -85,B 0,C 180,E1 -1516.333,E2 -1516.333} C_VEL
LIN {X 0,Y 587.423,Z 271.158,A -85,B 0,C 180,E1 -1516.509,E2 -1516.509} C_VEL
LIN {X 0,Y 587.864,Z 276.525,A -85,B 0,C 180,E1 -1516.585,E2 -1516.585} C_VEL
LIN {X 0,Y 587.724,Z 378.956,A -85,B 0,C 180,E1 -1517.855,E2 -1517.855} C_VEL
LIN {X 0,Y 587.676,Z 392.226,A -85,B 0,C 180,E1 -1518.161,E2 -1518.161} C_VEL
LIN {X 0,Y 587.595,Z 404.824,A -85,B 0,C 180,E1 -1518.592,E2 -1518.592} C_VEL
LIN {X 0,Y 587.554,Z 416.633,A -85,B 0,C 180,E1 -1519.141,E2 -1519.141} C_VEL
LIN {X 0,Y 587.453,Z 428.205,A -85,B 0,C 180,E1 -1519.836,E2 -1519.836} C_VEL
LIN {X 0,Y 587.393,Z 438.601,A -85,B 0,C 180,E1 -1520.618,E2 -1520.618} C_VEL
LIN {X 0,Y 587.321,Z 447.114,A -85,B 0,C 180,E1 -1521.398,E2 -1521.398} C_VEL
LIN {X 0,Y 587.274,Z 454.962,A -85,B 0,C 180,E1 -1522.263,E2 -1522.263} C_VEL
LIN {X 0,Y 587.23,Z 461.47,A -85,B 0,C 180,E1 -1523.126,E2 -1523.126} C_VEL
LIN {X 0,Y 587.236,Z 467.867,A -85,B 0,C 180,E1 -1524.162,E2 -1524.162} C_VEL
LIN {X 0,Y 587.147,Z 472.95,A -85,B 0,C 180,E1 -1525.194,E2 -1525.194} C_VEL
LIN {X 0,Y 587.213,Z 476.896,A -85,B 0,C 180,E1 -1526.226,E2 -1526.226} C_VEL
LIN {X 0,Y 587.132,Z 479.809,A -85,B 0,C 180,E1 -1527.256,E2 -1527.256} C_VEL
LIN {X 0,Y 587.14,Z 481.2,A -85,B 0,C 180,E1 -1527.942,E2 -1527.942} C_VEL
LIN {X 0,Y 587.14,Z 482.785,A -85,B 0,C 180,E1 -1529.314,E2 -1529.314} C_VEL
LIN {X 0,Y 587.137,Z 483,A -85,B 0,C 180,E1 -1530,E2 -1530} C_VEL
LIN {X 0,Y 587.147,Z 482.185,A -85,B 0,C 180,E1 -1531.372,E2 -1531.372} C_VEL
LIN {X 0,Y 587.14,Z 481.2,A -85,B 0,C 180,E1 -1532.058,E2 -1532.058} C_VEL
LIN {X 0,Y 587.132,Z 479.809,A -85,B 0,C 180,E1 -1532.744,E2 -1532.744} C_VEL
LIN {X 0,Y 587.213,Z 476.896,A -85,B 0,C 180,E1 -1533.774,E2 -1533.774} C_VEL
LIN {X 0,Y 587.147,Z 472.949,A -85,B 0,C 180,E1 -1534.806,E2 -1534.806} C_VEL
LIN {X 0,Y 587.217,Z 466.877,A -85,B 0,C 180,E1 -1536.011,E2 -1536.011} C_VEL
LIN {X 0,Y 587.245,Z 460.237,A -85,B 0,C 180,E1 -1537.046,E2 -1537.046} C_VEL
LIN {X 0,Y 587.3,Z 451.99,A -85,B 0,C 180,E1 -1538.083,E2 -1538.083} C_VEL
LIN {X 0,Y 587.343,Z 443.537,A -85,B 0,C 180,E1 -1538.949,E2 -1538.949} C_VEL
LIN {X 0,Y 587.419,Z 433.096,A -85,B 0,C 180,E1 -1539.816,E2 -1539.816} C_VEL
LIN {X 0,Y 587.508,Z 422.756,A -85,B 0,C 180,E1 -1540.511,E2 -1540.511} C_VEL
LIN {X 0,Y 587.568,Z 410.978,A -85,B 0,C 180,E1 -1541.141,E2 -1541.141} C_VEL
LIN {X 0,Y 587.61,Z 398.596,A -85,B 0,C 180,E1 -1541.64,E2 -1541.64} C_VEL
LIN {X 0,Y 587.69,Z 385.434,A -85,B 0,C 180,E1 -1542.014,E2 -1542.014} C_VEL
LIN {X 0,Y 587.718,Z 373.082,A -85,B 0,C 180,E1 -1542.233,E2 -1542.233} C_VEL
LIN {X 0,Y 587.701,Z 272.93,A -85,B 0,C 180,E1 -1543.463,E2 -1543.463} C_VEL
LIN {X 0,Y 587.379,Z 270.792,A -85,B 0,C 180,E1 -1543.515,E2 -1543.515} C_VEL
LIN {X 0,Y 587.481,Z 253.319,A -85,B 0,C 180,E1 -1545.971,E2 -1545.971} C_VEL
LIN {X 0,Y 587.596,Z 235.689,A -85,B 0,C 180,E1 -1548.479,E2 -1548.479} C_VEL
LIN {X 0,Y 587.721,Z 218.058,A -85,B 0,C 180,E1 -1551.023,E2 -1551.023} C_VEL
LIN {X 0,Y 587.813,Z 209.243,A -85,B 0,C 180,E1 -1552.309,E2 -1552.309} C_VEL
LIN {X 0,Y 587.319,Z 206.327,A -85,B 0,C 180,E1 -1552.788,E2 -1552.788} C_VEL
LIN {X 0,Y 587.331,Z 206.328,A -85,B 0,C 180,E1 -1555.517,E2 -1555.517} C_VEL
LIN {X 0,Y 587.338,Z 206.322,A -85,B 0,C 180,E1 -1557.818,E2 -1557.818} C_VEL
LIN {X 0,Y 587.323,Z 206.32,A -85,B 0,C 180,E1 -1560.507,E2 -1560.507} C_VEL
LIN {X 0,Y 587.335,Z 206.329,A -85,B 0,C 180,E1 -1563.396,E2 -1563.396} C_VEL
LIN {X 0,Y 587.29,Z 206.326,A -85,B 0,C 180,E1 -1565.9,E2 -1565.9} C_VEL
LIN {X 0,Y 587.321,Z 206.32,A -85,B 0,C 180,E1 -1568.48,E2 -1568.48} C_VEL
LIN {X 0,Y 587.336,Z 206.326,A -85,B 0,C 180,E1 -1571.157,E2 -1571.157} C_VEL
LIN {X 0,Y 587.32,Z 206.32,A -85,B 0,C 180,E1 -1574.112,E2 -1574.112} C_VEL
LIN {X 0,Y 587.313,Z 206.327,A -85,B 0,C 180,E1 -1576.993,E2 -1576.993} C_VEL
LIN {X 0,Y 587.313,Z 206.323,A -85,B 0,C 180,E1 -1579.745,E2 -1579.745} C_VEL
LIN {X 0,Y 587.343,Z 206.317,A -85,B 0,C 180,E1 -1582.392,E2 -1582.392} C_VEL
LIN {X 0,Y 587.33,Z 206.325,A -85,B 0,C 180,E1 -1584.944,E2 -1584.944} C_VEL
LIN {X 0,Y 587.336,Z 206.323,A -85,B 0,C 180,E1 -1587.421,E2 -1587.421} C_VEL
LIN {X 0,Y 587.333,Z 206.319,A -85,B 0,C 180,E1 -1589.83,E2 -1589.83} C_VEL
LIN {X 0,Y 587.351,Z 206.316,A -85,B 0,C 180,E1 -1592.307,E2 -1592.307} C_VEL
LIN {X 0,Y 587.35,Z 206.323,A -85,B 0,C 180,E1 -1595.241,E2 -1595.241} C_VEL
LIN {X 0,Y 587.32,Z 206.32,A -85,B 0,C 180,E1 -1598.226,E2 -1598.226} C_VEL
LIN {X 0,Y 587.347,Z 206.324,A -85,B 0,C 180,E1 -1601.151,E2 -1601.151} C_VEL
LIN {X 0,Y 587.323,Z 206.319,A -85,B 0,C 180,E1 -1604.025,E2 -1604.025} C_VEL
LIN {X 0,Y 587.36,Z 206.314,A -85,B 0,C 180,E1 -1606.154,E2 -1606.154} C_VEL
LIN {X 0,Y 587.339,Z 206.327,A -85,B 0,C 180,E1 -1608.962,E2 -1608.962} C_VEL
LIN {X 0,Y 587.364,Z 206.315,A -85,B 0,C 180,E1 -1611.745,E2 -1611.745} C_VEL
LIN {X 0,Y 587.364,Z 206.318,A -85,B 0,C 180,E1 -1614.507,E2 -1614.507} C_VEL
LIN {X 0,Y 587.366,Z 206.318,A -85,B 0,C 180,E1 -1617.257,E2 -1617.257} C_VEL
LIN {X 0,Y 587.383,Z 206.312,A -85,B 0,C 180,E1 -1620,E2 -1620} C_VEL
LIN {X 0,Y 587.373,Z 206.323,A -85,B 0,C 180,E1 -1622.743,E2 -1622.743} C_VEL
LIN {X 0,Y 587.353,Z 206.317,A -85,B 0,C 180,E1 -1625.493,E2 -1625.493} C_VEL
LIN {X 0,Y 587.369,Z 206.316,A -85,B 0,C 180,E1 -1628.255,E2 -1628.255} C_VEL
LIN {X 0,Y 587.347,Z 206.32,A -85,B 0,C 180,E1 -1631.134,E2 -1631.134} C_VEL
LIN {X 0,Y 587.364,Z 206.318,A -85,B 0,C 180,E1 -1634.261,E2 -1634.261} C_VEL
LIN {X 0,Y 587.346,Z 206.317,A -85,B 0,C 180,E1 -1637.406,E2 -1637.406} C_VEL
LIN {X 0,Y 587.308,Z 206.324,A -85,B 0,C 180,E1 -1638.313,E2 -1638.313} C_VEL
LIN {X 0,Y 586.666,Z 206.409,A -85,B 0,C 180,E1 -1638.885,E2 -1638.885} C_VEL
LIN {X 0,Y 583.842,Z 206.759,A -85,B 0,C 180,E1 -1639.814,E2 -1639.814} C_VEL
LIN {X 0,Y 581.431,Z 207.063,A -85,B 0,C 180,E1 -1640.561,E2 -1640.561} C_VEL
LIN {X 0,Y 580.377,Z 207.188,A -85,B 0,C 180,E1 -1641.137,E2 -1641.137} C_VEL
LIN {X 0,Y 580.281,Z 207.198,A -85,B 0,C 180,E1 -1641.332,E2 -1641.332} C_VEL
LIN {X 0,Y 580.297,Z 207.2,A -85,B 0,C 180,E1 -1644.317,E2 -1644.317} C_VEL
LIN {X 0,Y 580.263,Z 207.209,A -85,B 0,C 180,E1 -1646.624,E2 -1646.624} C_VEL
LIN {X 0,Y 580.296,Z 207.195,A -85,B 0,C 180,E1 -1649.309,E2 -1649.309} C_VEL
LIN {X 0,Y 580.297,Z 207.2,A -85,B 0,C 180,E1 -1652.201,E2 -1652.201} C_VEL
LIN {X 0,Y 580.279,Z 207.205,A -85,B 0,C 180,E1 -1654.697,E2 -1654.697} C_VEL
LIN {X 0,Y 580.274,Z 207.199,A -85,B 0,C 180,E1 -1657.271,E2 -1657.271} C_VEL
LIN {X 0,Y 580.287,Z 207.204,A -85,B 0,C 180,E1 -1660.27,E2 -1660.27} C_VEL
LIN {X 0,Y 580.271,Z 207.205,A -85,B 0,C 180,E1 -1662.707,E2 -1662.707} C_VEL
LIN {X 0,Y 580.322,Z 207.359,A -85,B 0,C 180,E1 -1665.38,E2 -1665.38} C_VEL
LIN {X 0,Y 580.516,Z 212.946,A -85,B 0,C 180,E1 -1666.365,E2 -1666.365} C_VEL
LIN {X 0,Y 580.351,Z 227.66,A -85,B 0,C 180,E1 -1668.911,E2 -1668.911} C_VEL
LIN {X 0,Y 580.282,Z 242.154,A -85,B 0,C 180,E1 -1671.39,E2 -1671.39} C_VEL
LIN {X 0,Y 580.987,Z 247.51,A -85,B 0,C 180,E1 -1671.481,E2 -1671.481} C_VEL
LIN {X 0,Y 580.748,Z 349.644,A -85,B 0,C 180,E1 -1672.765,E2 -1672.765} C_VEL
LIN {X 0,Y 580.716,Z 363.217,A -85,B 0,C 180,E1 -1673.091,E2 -1673.091} C_VEL
LIN {X 0,Y 580.63,Z 375.428,A -85,B 0,C 180,E1 -1673.522,E2 -1673.522} C_VEL
LIN {X 0,Y 580.517,Z 387.704,A -85,B 0,C 180,E1 -1674.113,E2 -1674.113} C_VEL
LIN {X 0,Y 580.42,Z 398.595,A -85,B 0,C 180,E1 -1674.784,E2 -1674.784} C_VEL
LIN {X 0,Y 580.37,Z 408.969,A -85,B 0,C 180,E1 -1675.579,E2 -1675.579} C_VEL
LIN {X 0,Y 580.257,Z 418.199,A -85,B 0,C 180,E1 -1676.449,E2 -1676.449} C_VEL
LIN {X 0,Y 580.23,Z 426.302,A -85,B 0,C 180,E1 -1677.384,E2 -1677.384} C_VEL
LIN {X 0,Y 580.19,Z 432.864,A -85,B 0,C 180,E1 -1678.3,E2 -1678.3} C_VEL
LIN {X 0,Y 580.127,Z 439.327,A -85,B 0,C 180,E1 -1679.415,E2 -1679.415} C_VEL
LIN {X 0,Y 580.111,Z 444.261,A -85,B 0,C 180,E1 -1680.501,E2 -1680.501} C_VEL
LIN {X 0,Y 580.056,Z 448.624,A -85,B 0,C 180,E1 -1681.802,E2 -1681.802} C_VEL
LIN {X 0,Y 580.062,Z 450.485,A -85,B 0,C 180,E1 -1682.587,E2 -1682.587} C_VEL
LIN {X 0,Y 580.047,Z 452.253,A -85,B 0,C 180,E1 -1683.716,E2 -1683.716} C_VEL
LIN {X 0,Y 580.01,Z 452.975,A -85,B 0,C 180,E1 -1684.907,E2 -1684.907} C_VEL
LIN {X 0,Y 580.013,Z 452.831,A -85,B 0,C 180,E1 -1685.671,E2 -1685.671} C_VEL
LIN {X 0,Y 580.049,Z 451.327,A -85,B 0,C 180,E1 -1687.049,E2 -1687.049} C_VEL
LIN {X 0,Y 580.079,Z 448.557,A -85,B 0,C 180,E1 -1688.314,E2 -1688.314} C_VEL
LIN {X 0,Y 580.097,Z 444.898,A -85,B 0,C 180,E1 -1689.431,E2 -1689.431} C_VEL
LIN {X 0,Y 580.136,Z 440.023,A -85,B 0,C 180,E1 -1690.541,E2 -1690.541} C_VEL
LIN {X 0,Y 580.18,Z 433.809,A -85,B 0,C 180,E1 -1691.642,E2 -1691.642} C_VEL
LIN {X 0,Y 580.201,Z 426.068,A -85,B 0,C 180,E1 -1692.736,E2 -1692.736} C_VEL
LIN {X 0,Y 580.278,Z 418.159,A -85,B 0,C 180,E1 -1693.645,E2 -1693.645} C_VEL
LIN {X 0,Y 580.312,Z 408.54,A -85,B 0,C 180,E1 -1694.548,E2 -1694.548} C_VEL
LIN {X 0,Y 580.421,Z 397.915,A -85,B 0,C 180,E1 -1695.353,E2 -1695.353} C_VEL
LIN {X 0,Y 580.533,Z 387.502,A -85,B 0,C 180,E1 -1695.988,E2 -1695.988} C_VEL
LIN {X 0,Y 580.631,Z 375.357,A -85,B 0,C 180,E1 -1696.571,E2 -1696.571} C_VEL
LIN {X 0,Y 580.694,Z 362.623,A -85,B 0,C 180,E1 -1697.017,E2 -1697.017} C_VEL
LIN {X 0,Y 580.742,Z 349.398,A -85,B 0,C 180,E1 -1697.329,E2 -1697.329} C_VEL
LIN {X 0,Y 580.862,Z 245.692,A -85,B 0,C 180,E1 -1698.635,E2 -1698.635} C_VEL
LIN {X 0,Y 580.285,Z 242.153,A -85,B 0,C 180,E1 -1698.7,E2 -1698.7} C_VEL
LIN {X 0,Y 580.392,Z 226.988,A -85,B 0,C 180,E1 -1701.294,E2 -1701.294} C_VEL
LIN {X 0,Y 580.529,Z 211.833,A -85,B 0,C 180,E1 -1703.919,E2 -1703.919} C_VEL
LIN {X 0,Y 580.287,Z 207.202,A -85,B 0,C 180,E1 -1704.745,E2 -1704.745} C_VEL
LIN {X 0,Y 580.34,Z 207.196,A -85,B 0,C 180,E1 -1707.918,E2 -1707.918} C_VEL
LIN {X 0,Y 580.351,Z 207.193,A -85,B 0,C 180,E1 -1710,E2 -1710} C_VEL
LIN {X 0,Y 580.311,Z 207.193,A -85,B 0,C 180,E1 -1712.777,E2 -1712.777} C_VEL
LIN {X 0,Y 580.311,Z 207.202,A -85,B 0,C 180,E1 -1715.56,E2 -1715.56} C_VEL
LIN {X 0,Y 580.307,Z 207.194,A -85,B 0,C 180,E1 -1718.356,E2 -1718.356} C_VEL
LIN {X 0,Y 580.305,Z 207.198,A -85,B 0,C 180,E1 -1721.191,E2 -1721.191} C_VEL
LIN {X 0,Y 580.3,Z 207.195,A -85,B 0,C 180,E1 -1724.331,E2 -1724.331} C_VEL
LIN {X 0,Y 580.27,Z 207.2,A -85,B 0,C 180,E1 -1726.898,E2 -1726.898} C_VEL
LIN {X 0,Y 580.282,Z 207.202,A -85,B 0,C 180,E1 -1729.823,E2 -1729.823} C_VEL
LIN {X 0,Y 580.256,Z 207.202,A -85,B 0,C 180,E1 -1732.053,E2 -1732.053} C_VEL
LIN {X 0,Y 580.289,Z 207.2,A -85,B 0,C 180,E1 -1735.08,E2 -1735.08} C_VEL
LIN {X 0,Y 580.291,Z 207.197,A -85,B 0,C 180,E1 -1738.186,E2 -1738.186} C_VEL
LIN {X 0,Y 580.273,Z 207.199,A -85,B 0,C 180,E1 -1740.692,E2 -1740.692} C_VEL
LIN {X 0,Y 580.304,Z 207.203,A -85,B 0,C 180,E1 -1743.316,E2 -1743.316} C_VEL
LIN {X 0,Y 580.243,Z 207.206,A -85,B 0,C 180,E1 -1745.755,E2 -1745.755} C_VEL
LIN {X 0,Y 580.285,Z 207.197,A -85,B 0,C 180,E1 -1748.146,E2 -1748.146} C_VEL
LIN {X 0,Y 580.296,Z 207.198,A -85,B 0,C 180,E1 -1750.843,E2 -1750.843} C_VEL
LIN {X 0,Y 580.27,Z 207.204,A -85,B 0,C 180,E1 -1753.658,E2 -1753.658} C_VEL
LIN {X 0,Y 580.275,Z 207.199,A -85,B 0,C 180,E1 -1756.609,E2 -1756.609} C_VEL
LIN {X 0,Y 580.295,Z 207.203,A -85,B 0,C 180,E1 -1759.156,E2 -1759.156} C_VEL
LIN {X 0,Y 580.288,Z 207.198,A -85,B 0,C 180,E1 -1761.927,E2 -1761.927} C_VEL
LIN {X 0,Y 580.285,Z 207.197,A -85,B 0,C 180,E1 -1764.455,E2 -1764.455} C_VEL
LIN {X 0,Y 580.288,Z 207.202,A -85,B 0,C 180,E1 -1766.975,E2 -1766.975} C_VEL
LIN {X 0,Y 580.294,Z 207.203,A -85,B 0,C 180,E1 -1769.425,E2 -1769.425} C_VEL
LIN {X 0,Y 580.296,Z 207.196,A -85,B 0,C 180,E1 -1772.141,E2 -1772.141} C_VEL
LIN {X 0,Y 580.319,Z 207.202,A -85,B 0,C 180,E1 -1775.269,E2 -1775.269} C_VEL
LIN {X 0,Y 580.27,Z 207.199,A -85,B 0,C 180,E1 -1777.947,E2 -1777.947} C_VEL
LIN {X 0,Y 580.296,Z 207.202,A -85,B 0,C 180,E1 -1780.913,E2 -1780.913} C_VEL
LIN {X 0,Y 580.276,Z 207.199,A -85,B 0,C 180,E1 -1783.825,E2 -1783.825} C_VEL
LIN {X 0,Y 580.323,Z 207.192,A -85,B 0,C 180,E1 -1785.983,E2 -1785.983} C_VEL
LIN {X 0,Y 580.302,Z 207.201,A -85,B 0,C 180,E1 -1788.827,E2 -1788.827} C_VEL
LIN {X 0,Y 580.331,Z 207.193,A -85,B 0,C 180,E1 -1791.644,E2 -1791.644} C_VEL
LIN {X 0,Y 580.327,Z 207.193,A -85,B 0,C 180,E1 -1794.44,E2 -1794.44} C_VEL
LIN {X 0,Y 580.336,Z 207.198,A -85,B 0,C 180,E1 -1797.223,E2 -1797.223} C_VEL
LIN {X 0,Y 580.351,Z 207.189,A -85,B 0,C 180,E1 -1800,E2 -1800} C_VEL
LIN {X 0,Y 580.335,Z 207.197,A -85,B 0,C 180,E1 -1802.777,E2 -1802.777} C_VEL
LIN {X 0,Y 580.328,Z 207.193,A -85,B 0,C 180,E1 -1805.56,E2 -1805.56} C_VEL
LIN {X 0,Y 580.326,Z 207.193,A -85,B 0,C 180,E1 -1808.356,E2 -1808.356} C_VEL
LIN {X 0,Y 580.297,Z 207.201,A -85,B 0,C 180,E1 -1811.191,E2 -1811.191} C_VEL
LIN {X 0,Y 580.323,Z 207.192,A -85,B 0,C 180,E1 -1814.017,E2 -1814.017} C_VEL
LIN {X 0,Y 580.309,Z 207.203,A -85,B 0,C 180,E1 -1816.914,E2 -1816.914} C_VEL
LIN {X 0,Y 580.302,Z 207.195,A -85,B 0,C 180,E1 -1819.822,E2 -1819.822} C_VEL
LIN {X 0,Y 580.292,Z 207.206,A -85,B 0,C 180,E1 -1822.803,E2 -1822.803} C_VEL
LIN {X 0,Y 580.302,Z 207.201,A -85,B 0,C 180,E1 -1825.08,E2 -1825.08} C_VEL
LIN {X 0,Y 580.298,Z 207.197,A -85,B 0,C 180,E1 -1828.186,E2 -1828.186} C_VEL
LIN {X 0,Y 580.282,Z 207.206,A -85,B 0,C 180,E1 -1830.695,E2 -1830.695} C_VEL
LIN {X 0,Y 580.3,Z 207.197,A -85,B 0,C 180,E1 -1833.316,E2 -1833.316} C_VEL
LIN {X 0,Y 580.275,Z 207.198,A -85,B 0,C 180,E1 -1835.761,E2 -1835.761} C_VEL
LIN {X 0,Y 580.286,Z 207.198,A -85,B 0,C 180,E1 -1838.147,E2 -1838.147} C_VEL
LIN {X 0,Y 580.295,Z 207.204,A -85,B 0,C 180,E1 -1840.844,E2 -1840.844} C_VEL
LIN {X 0,Y 580.277,Z 207.198,A -85,B 0,C 180,E1 -1843.658,E2 -1843.658} C_VEL
LIN {X 0,Y 580.28,Z 207.207,A -85,B 0,C 180,E1 -1846.609,E2 -1846.609} C_VEL
LIN {X 0,Y 580.296,Z 207.198,A -85,B 0,C 180,E1 -1849.157,E2 -1849.157} C_VEL
LIN {X 0,Y 580.287,Z 207.197,A -85,B 0,C 180,E1 -1851.928,E2 -1851.928} C_VEL
LIN {X 0,Y 580.249,Z 207.208,A -85,B 0,C 180,E1 -1854.453,E2 -1854.453} C_VEL
LIN {X 0,Y 580.288,Z 207.2,A -85,B 0,C 180,E1 -1856.975,E2 -1856.975} C_VEL
LIN {X 0,Y 580.291,Z 207.196,A -85,B 0,C 180,E1 -1859.425,E2 -1859.425} C_VEL
LIN {X 0,Y 580.289,Z 207.2,A -85,B 0,C 180,E1 -1862.144,E2 -1862.144} C_VEL
LIN {X 0,Y 580.289,Z 207.202,A -85,B 0,C 180,E1 -1864.92,E2 -1864.92} C_VEL
LIN {X 0,Y 580.265,Z 207.238,A -85,B 0,C 180,E1 -1867.107,E2 -1867.107} C_VEL
LIN {X 0,Y 580.908,Z 211.695,A -85,B 0,C 180,E1 -1867.786,E2 -1867.786} C_VEL
LIN {X 0,Y 580.702,Z 230.407,A -85,B 0,C 180,E1 -1870.524,E2 -1870.524} C_VEL
LIN {X 0,Y 580.536,Z 249.543,A -85,B 0,C 180,E1 -1873.291,E2 -1873.291} C_VEL
LIN {X 0,Y 580.389,Z 270.794,A -85,B 0,C 180,E1 -1876.32,E2 -1876.32} C_VEL
LIN {X 0,Y 580.966,Z 276.525,A -85,B 0,C 180,E1 -1876.423,E2 -1876.423} C_VEL
LIN {X 0,Y 580.807,Z 378.956,A -85,B 0,C 180,E1 -1877.708,E2 -1877.708} C_VEL
LIN {X 0,Y 580.735,Z 392.226,A -85,B 0,C 180,E1 -1878.017,E2 -1878.017} C_VEL
LIN {X 0,Y 580.63,Z 404.379,A -85,B 0,C 180,E1 -1878.436,E2 -1878.436} C_VEL
LIN {X 0,Y 580.557,Z 416.631,A -85,B 0,C 180,E1 -1879.009,E2 -1879.009} C_VEL
LIN {X 0,Y 580.428,Z 428.204,A -85,B 0,C 180,E1 -1879.712,E2 -1879.712} C_VEL
LIN {X 0,Y 580.344,Z 438.602,A -85,B 0,C 180,E1 -1880.503,E2 -1880.503} C_VEL
LIN {X 0,Y 580.271,Z 447.114,A -85,B 0,C 180,E1 -1881.292,E2 -1881.292} C_VEL
LIN {X 0,Y 580.222,Z 454.962,A -85,B 0,C 180,E1 -1882.168,E2 -1882.168} C_VEL
LIN {X 0,Y 580.153,Z 462.651,A -85,B 0,C 180,E1 -1883.222,E2 -1883.222} C_VEL
LIN {X 0,Y 580.139,Z 469.681,A -85,B 0,C 180,E1 -1884.439,E2 -1884.439} C_VEL
LIN {X 0,Y 580.108,Z 474.372,A -85,B 0,C 180,E1 -1885.484,E2 -1885.484} C_VEL
LIN {X 0,Y 580.123,Z 477.958,A -85,B 0,C 180,E1 -1886.527,E2 -1886.527} C_VEL
LIN {X 0,Y 580.043,Z 479.809,A -85,B 0,C 180,E1 -1887.222,E2 -1887.222} C_VEL
LIN {X 0,Y 580.039,Z 481.199,A -85,B 0,C 180,E1 -1887.917,E2 -1887.917} C_VEL
LIN {X 0,Y 580.04,Z 482.785,A -85,B 0,C 180,E1 -1889.306,E2 -1889.306} C_VEL
LIN {X 0,Y 580.037,Z 483,A -85,B 0,C 180,E1 -1890,E2 -1890} C_VEL
LIN {X 0,Y 580.046,Z 482.186,A -85,B 0,C 180,E1 -1891.389,E2 -1891.389} C_VEL
LIN {X 0,Y 580.039,Z 481.2,A -85,B 0,C 180,E1 -1892.083,E2 -1892.083} C_VEL
LIN {X 0,Y 580.043,Z 479.81,A -85,B 0,C 180,E1 -1892.778,E2 -1892.778} C_VEL
LIN {X 0,Y 580.11,Z 476.896,A -85,B 0,C 180,E1 -1893.821,E2 -1893.821} C_VEL
LIN {X 0,Y 580.053,Z 472.949,A -85,B 0,C 180,E1 -1894.865,E2 -1894.865} C_VEL
LIN {X 0,Y 580.139,Z 466.876,A -85,B 0,C 180,E1 -1896.085,E2 -1896.085} C_VEL
LIN {X 0,Y 580.184,Z 460.237,A -85,B 0,C 180,E1 -1897.132,E2 -1897.132} C_VEL
LIN {X 0,Y 580.25,Z 451.99,A -85,B 0,C 180,E1 -1898.182,E2 -1898.182} C_VEL
LIN {X 0,Y 580.308,Z 443.538,A -85,B 0,C 180,E1 -1899.058,E2 -1899.058} C_VEL
LIN {X 0,Y 580.419,Z 433.097,A -85,B 0,C 180,E1 -1899.936,E2 -1899.936} C_VEL
LIN {X 0,Y 580.512,Z 422.754,A -85,B 0,C 180,E1 -1900.639,E2 -1900.639} C_VEL
LIN {X 0,Y 580.581,Z 411.407,A -85,B 0,C 180,E1 -1901.256,E2 -1901.256} C_VEL
LIN {X 0,Y 580.654,Z 399.766,A -85,B 0,C 180,E1 -1901.741,E2 -1901.741} C_VEL
LIN {X 0,Y 580.729,Z 386.347,A -85,B 0,C 180,E1 -1902.138,E2 -1902.138} C_VEL
LIN {X 0,Y 580.79,Z 373.082,A -85,B 0,C 180,E1 -1902.381,E2 -1902.381} C_VEL
LIN {X 0,Y 580.787,Z 273.601,A -85,B 0,C 180,E1 -1903.618,E2 -1903.618} C_VEL
LIN {X 0,Y 580.389,Z 270.792,A -85,B 0,C 180,E1 -1903.68,E2 -1903.68} C_VEL
LIN {X 0,Y 580.536,Z 249.541,A -85,B 0,C 180,E1 -1906.709,E2 -1906.709} C_VEL
LIN {X 0,Y 580.703,Z 230.406,A -85,B 0,C 180,E1 -1909.476,E2 -1909.476} C_VEL
LIN {X 0,Y 580.908,Z 211.668,A -85,B 0,C 180,E1 -1912.214,E2 -1912.214} C_VEL
LIN {X 0,Y 580.272,Z 207.206,A -85,B 0,C 180,E1 -1912.923,E2 -1912.923} C_VEL
LIN {X 0,Y 580.29,Z 207.202,A -85,B 0,C 180,E1 -1915.08,E2 -1915.08} C_VEL
LIN {X 0,Y 580.292,Z 207.197,A -85,B 0,C 180,E1 -1918.186,E2 -1918.186} C_VEL
LIN {X 0,Y 580.274,Z 207.199,A -85,B 0,C 180,E1 -1920.692,E2 -1920.692} C_VEL
LIN {X 0,Y 580.304,Z 207.204,A -85,B 0,C 180,E1 -1923.316,E2 -1923.316} C_VEL
LIN {X 0,Y 580.244,Z 207.205,A -85,B 0,C 180,E1 -1925.756,E2 -1925.756} C_VEL
LIN {X 0,Y 580.286,Z 207.197,A -85,B 0,C 180,E1 -1928.146,E2 -1928.146} C_VEL
LIN {X 0,Y 580.297,Z 207.198,A -85,B 0,C 180,E1 -1930.843,E2 -1930.843} C_VEL
LIN {X 0,Y 580.282,Z 207.201,A -85,B 0,C 180,E1 -1933.657,E2 -1933.657} C_VEL
LIN {X 0,Y 580.276,Z 207.199,A -85,B 0,C 180,E1 -1936.609,E2 -1936.609} C_VEL
LIN {X 0,Y 580.297,Z 207.204,A -85,B 0,C 180,E1 -1939.156,E2 -1939.156} C_VEL
LIN {X 0,Y 580.29,Z 207.196,A -85,B 0,C 180,E1 -1941.927,E2 -1941.927} C_VEL
LIN {X 0,Y 580.287,Z 207.197,A -85,B 0,C 180,E1 -1944.455,E2 -1944.455} C_VEL
LIN {X 0,Y 580.289,Z 207.203,A -85,B 0,C 180,E1 -1946.975,E2 -1946.975} C_VEL
LIN {X 0,Y 580.296,Z 207.2,A -85,B 0,C 180,E1 -1949.425,E2 -1949.425} C_VEL
LIN {X 0,Y 580.297,Z 207.194,A -85,B 0,C 180,E1 -1952.141,E2 -1952.141} C_VEL
LIN {X 0,Y 580.321,Z 207.198,A -85,B 0,C 180,E1 -1955.27,E2 -1955.27} C_VEL
LIN {X 0,Y 580.271,Z 207.198,A -85,B 0,C 180,E1 -1957.947,E2 -1957.947} C_VEL
LIN {X 0,Y 580.296,Z 207.204,A -85,B 0,C 180,E1 -1960.913,E2 -1960.913} C_VEL
LIN {X 0,Y 580.276,Z 207.198,A -85,B 0,C 180,E1 -1963.825,E2 -1963.825} C_VEL
LIN {X 0,Y 580.326,Z 207.19,A -85,B 0,C 180,E1 -1965.983,E2 -1965.983} C_VEL
LIN {X 0,Y 580.304,Z 207.202,A -85,B 0,C 180,E1 -1968.827,E2 -1968.827} C_VEL
LIN {X 0,Y 580.327,Z 207.192,A -85,B 0,C 180,E1 -1971.644,E2 -1971.644} C_VEL
LIN {X 0,Y 580.33,Z 207.194,A -85,B 0,C 180,E1 -1974.44,E2 -1974.44} C_VEL
LIN {X 0,Y 580.333,Z 207.195,A -85,B 0,C 180,E1 -1977.223,E2 -1977.223} C_VEL
LIN {X 0,Y 580.352,Z 207.187,A -85,B 0,C 180,E1 -1980,E2 -1980} C_VEL
LIN {X 0,Y 580.338,Z 207.2,A -85,B 0,C 180,E1 -1982.777,E2 -1982.777} C_VEL
LIN {X 0,Y 580.322,Z 207.192,A -85,B 0,C 180,E1 -1985.56,E2 -1985.56} C_VEL
LIN {X 0,Y 580.332,Z 207.194,A -85,B 0,C 180,E1 -1988.356,E2 -1988.356} C_VEL
LIN {X 0,Y 580.299,Z 207.197,A -85,B 0,C 180,E1 -1991.191,E2 -1991.191} C_VEL
LIN {X 0,Y 580.323,Z 207.193,A -85,B 0,C 180,E1 -1994.017,E2 -1994.017} C_VEL
LIN {X 0,Y 580.312,Z 207.199,A -85,B 0,C 180,E1 -1996.914,E2 -1996.914} C_VEL
LIN {X 0,Y 580.286,Z 207.197,A -85,B 0,C 180,E1 -1999.823,E2 -1999.823} C_VEL
LIN {X 0,Y 580.281,Z 207.198,A -85,B 0,C 180,E1 -2001.332,E2 -2001.332} C_VEL
LIN {X 0,Y 579.582,Z 207.285,A -85,B 0,C 180,E1 -2001.912,E2 -2001.912} C_VEL
LIN {X 0,Y 576.704,Z 207.648,A -85,B 0,C 180,E1 -2002.851,E2 -2002.851} C_VEL
LIN {X 0,Y 574.31,Z 207.943,A -85,B 0,C 180,E1 -2003.608,E2 -2003.608} C_VEL
LIN {X 0,Y 573.312,Z 208.069,A -85,B 0,C 180,E1 -2004.191,E2 -2004.191} C_VEL
LIN {X 0,Y 573.246,Z 208.079,A -85,B 0,C 180,E1 -2004.389,E2 -2004.389} C_VEL
LIN {X 0,Y 573.2,Z 208.083,A -85,B 0,C 180,E1 -2006.979,E2 -2006.979} C_VEL
LIN {X 0,Y 573.242,Z 208.073,A -85,B 0,C 180,E1 -2009.488,E2 -2009.488} C_VEL
LIN {X 0,Y 573.252,Z 208.081,A -85,B 0,C 180,E1 -2012.645,E2 -2012.645} C_VEL
LIN {X 0,Y 573.193,Z 208.082,A -85,B 0,C 180,E1 -2015.189,E2 -2015.189} C_VEL
LIN {X 0,Y 573.222,Z 208.078,A -85,B 0,C 180,E1 -2017.809,E2 -2017.809} C_VEL
LIN {X 0,Y 573.245,Z 208.083,A -85,B 0,C 180,E1 -2020.525,E2 -2020.525} C_VEL
LIN {X 0,Y 573.207,Z 208.08,A -85,B 0,C 180,E1 -2023.362,E2 -2023.362} C_VEL
LIN {X 0,Y 573.283,Z 208.251,A -85,B 0,C 180,E1 -2025.319,E2 -2025.319} C_VEL
LIN {X 0,Y 573.549,Z 212.401,A -85,B 0,C 180,E1 -2026.035,E2 -2026.035} C_VEL
LIN {X 0,Y 573.349,Z 226.776,A -85,B 0,C 180,E1 -2028.554,E2 -2028.554} C_VEL
LIN {X 0,Y 573.275,Z 242.108,A -85,B 0,C 180,E1 -2031.212,E2 -2031.212} C_VEL
LIN {X 0,Y 574.086,Z 248.279,A -85,B 0,C 180,E1 -2031.324,E2 -2031.324} C_VEL
LIN {X 0,Y 573.808,Z 348.914,A -85,B 0,C 180,E1 -2032.6,E2 -2032.6} C_VEL
LIN {X 0,Y 573.757,Z 362.116,A -85,B 0,C 180,E1 -2032.911,E2 -2032.911} C_VEL
LIN {X 0,Y 573.685,Z 374.134,A -85,B 0,C 180,E1 -2033.329,E2 -2033.329} C_VEL
LIN {X 0,Y 573.575,Z 385.672,A -85,B 0,C 180,E1 -2033.866,E2 -2033.866} C_VEL
LIN {X 0,Y 573.453,Z 396.413,A -85,B 0,C 180,E1 -2034.507,E2 -2034.507} C_VEL
LIN {X 0,Y 573.349,Z 407.57,A -85,B 0,C 180,E1 -2035.344,E2 -2035.344} C_VEL
LIN {X 0,Y 573.255,Z 416.825,A -85,B 0,C 180,E1 -2036.201,E2 -2036.201} C_VEL
LIN {X 0,Y 573.12,Z 425.14,A -85,B 0,C 180,E1 -2037.138,E2 -2037.138} C_VEL
LIN {X 0,Y 573.117,Z 432.614,A -85,B 0,C 180,E1 -2038.177,E2 -2038.177} C_VEL
LIN {X 0,Y 573.059,Z 438.307,A -85,B 0,C 180,E1 -2039.147,E2 -2039.147} C_VEL
LIN {X 0,Y 573.018,Z 443.316,A -85,B 0,C 180,E1 -2040.211,E2 -2040.211} C_VEL
LIN {X 0,Y 572.973,Z 447.636,A -85,B 0,C 180,E1 -2041.421,E2 -2041.421} C_VEL
LIN {X 0,Y 572.966,Z 449.775,A -85,B 0,C 180,E1 -2042.218,E2 -2042.218} C_VEL
LIN {X 0,Y 572.956,Z 452.101,A -85,B 0,C 180,E1 -2043.565,E2 -2043.565} C_VEL
LIN {X 0,Y 572.935,Z 452.901,A -85,B 0,C 180,E1 -2044.575,E2 -2044.575} C_VEL
LIN {X 0,Y 572.932,Z 452.938,A -85,B 0,C 180,E1 -2045.35,E2 -2045.35} C_VEL
LIN {X 0,Y 572.92,Z 452.533,A -85,B 0,C 180,E1 -2046.121,E2 -2046.121} C_VEL
LIN {X 0,Y 572.955,Z 451.565,A -85,B 0,C 180,E1 -2046.922,E2 -2046.922} C_VEL
LIN {X 0,Y 572.947,Z 450.243,A -85,B 0,C 180,E1 -2047.65,E2 -2047.65} C_VEL
LIN {X 0,Y 572.989,Z 447.304,A -85,B 0,C 180,E1 -2048.778,E2 -2048.778} C_VEL
LIN {X 0,Y 573.029,Z 443.171,A -85,B 0,C 180,E1 -2049.915,E2 -2049.915} C_VEL
LIN {X 0,Y 573.074,Z 437.49,A -85,B 0,C 180,E1 -2051.098,E2 -2051.098} C_VEL
LIN {X 0,Y 573.121,Z 431.058,A -85,B 0,C 180,E1 -2052.148,E2 -2052.148} C_VEL
LIN {X 0,Y 573.176,Z 423.764,A -85,B 0,C 180,E1 -2053.117,E2 -2053.117} C_VEL
LIN {X 0,Y 573.267,Z 414.005,A -85,B 0,C 180,E1 -2054.171,E2 -2054.171} C_VEL
LIN {X 0,Y 573.363,Z 404.554,A -85,B 0,C 180,E1 -2054.993,E2 -2054.993} C_VEL
LIN {X 0,Y 573.462,Z 394.215,A -85,B 0,C 180,E1 -2055.725,E2 -2055.725} C_VEL
LIN {X 0,Y 573.635,Z 383.001,A -85,B 0,C 180,E1 -2056.359,E2 -2056.359} C_VEL
LIN {X 0,Y 573.694,Z 370.595,A -85,B 0,C 180,E1 -2056.901,E2 -2056.901} C_VEL
LIN {X 0,Y 573.761,Z 357.39,A -85,B 0,C 180,E1 -2057.308,E2 -2057.308} C_VEL
LIN {X 0,Y 573.839,Z 344.559,A -85,B 0,C 180,E1 -2057.556,E2 -2057.556} C_VEL
LIN {X 0,Y 573.92,Z 246.097,A -85,B 0,C 180,E1 -2058.798,E2 -2058.798} C_VEL
LIN {X 0,Y 573.247,Z 242.093,A -85,B 0,C 180,E1 -2058.881,E2 -2058.881} C_VEL
LIN {X 0,Y 573.377,Z 227.756,A -85,B 0,C 180,E1 -2061.364,E2 -2061.364} C_VEL
LIN {X 0,Y 573.535,Z 212.601,A -85,B 0,C 180,E1 -2064.021,E2 -2064.021} C_VEL
LIN {X 0,Y 573.271,Z 208.077,A -85,B 0,C 180,E1 -2064.857,E2 -2064.857} C_VEL
LIN {X 0,Y 573.31,Z 208.073,A -85,B 0,C 180,E1 -2067.892,E2 -2067.892} C_VEL
LIN {X 0,Y 573.32,Z 208.069,A -85,B 0,C 180,E1 -2070,E2 -2070} C_VEL
LIN {X 0,Y 573.28,Z 208.069,A -85,B 0,C 180,E1 -2072.811,E2 -2072.811} C_VEL
LIN {X 0,Y 573.279,Z 208.079,A -85,B 0,C 180,E1 -2075.628,E2 -2075.628} C_VEL
LIN {X 0,Y 573.25,Z 208.073,A -85,B 0,C 180,E1 -2078.46,E2 -2078.46} C_VEL
LIN {X 0,Y 573.276,Z 208.075,A -85,B 0,C 180,E1 -2081.312,E2 -2081.312} C_VEL
LIN {X 0,Y 573.274,Z 208.07,A -85,B 0,C 180,E1 -2084.42,E2 -2084.42} C_VEL
LIN {X 0,Y 573.241,Z 208.078,A -85,B 0,C 180,E1 -2087.112,E2 -2087.112} C_VEL
LIN {X 0,Y 573.237,Z 208.077,A -85,B 0,C 180,E1 -2090.077,E2 -2090.077} C_VEL
LIN {X 0,Y 573.223,Z 208.077,A -85,B 0,C 180,E1 -2092.338,E2 -2092.338} C_VEL
LIN {X 0,Y 573.236,Z 208.083,A -85,B 0,C 180,E1 -2095.411,E2 -2095.411} C_VEL
LIN {X 0,Y 573.23,Z 208.076,A -85,B 0,C 180,E1 -2098.565,E2 -2098.565} C_VEL
LIN {X 0,Y 573.22,Z 208.08,A -85,B 0,C 180,E1 -2100.993,E2 -2100.993} C_VEL
LIN {X 0,Y 573.264,Z 208.08,A -85,B 0,C 180,E1 -2103.524,E2 -2103.524} C_VEL
LIN {X 0,Y 573.193,Z 208.082,A -85,B 0,C 180,E1 -2106.053,E2 -2106.053} C_VEL
LIN {X 0,Y 573.238,Z 208.076,A -85,B 0,C 180,E1 -2108.701,E2 -2108.701} C_VEL
LIN {X 0,Y 573.227,Z 208.082,A -85,B 0,C 180,E1 -2111.592,E2 -2111.592} C_VEL
LIN {X 0,Y 573.224,Z 208.076,A -85,B 0,C 180,E1 -2114.334,E2 -2114.334} C_VEL
LIN {X 0,Y 573.239,Z 208.084,A -85,B 0,C 180,E1 -2117.358,E2 -2117.358} C_VEL
LIN {X 0,Y 573.237,Z 208.075,A -85,B 0,C 180,E1 -2120.392,E2 -2120.392} C_VEL
LIN {X 0,Y 573.254,Z 208.08,A -85,B 0,C 180,E1 -2123.077,E2 -2123.077} C_VEL
LIN {X 0,Y 573.268,Z 208.075,A -85,B 0,C 180,E1 -2125.671,E2 -2125.671} C_VEL
LIN {X 0,Y 573.238,Z 208.075,A -85,B 0,C 180,E1 -2128.184,E2 -2128.184} C_VEL
LIN {X 0,Y 573.263,Z 208.074,A -85,B 0,C 180,E1 -2130.634,E2 -2130.634} C_VEL
LIN {X 0,Y 573.248,Z 208.081,A -85,B 0,C 180,E1 -2133.024,E2 -2133.024} C_VEL
LIN {X 0,Y 573.273,Z 208.078,A -85,B 0,C 180,E1 -2135.366,E2 -2135.366} C_VEL
LIN {X 0,Y 573.226,Z 208.077,A -85,B 0,C 180,E1 -2138.419,E2 -2138.419} C_VEL
LIN {X 0,Y 573.266,Z 208.075,A -85,B 0,C 180,E1 -2140.731,E2 -2140.731} C_VEL
LIN {X 0,Y 573.248,Z 208.076,A -85,B 0,C 180,E1 -2143.622,E2 -2143.622} C_VEL
LIN {X 0,Y 573.271,Z 208.072,A -85,B 0,C 180,E1 -2145.807,E2 -2145.807} C_VEL
LIN {X 0,Y 573.26,Z 208.077,A -85,B 0,C 180,E1 -2148.745,E2 -2148.745} C_VEL
LIN {X 0,Y 573.287,Z 208.072,A -85,B 0,C 180,E1 -2151.54,E2 -2151.54} C_VEL
LIN {X 0,Y 573.295,Z 208.069,A -85,B 0,C 180,E1 -2154.372,E2 -2154.372} C_VEL
LIN {X 0,Y 573.312,Z 208.066,A -85,B 0,C 180,E1 -2157.892,E2 -2157.892} C_VEL
LIN {X 0,Y 573.327,Z 208.069,A -85,B 0,C 180,E1 -2160.702,E2 -2160.702} C_VEL
LIN {X 0,Y 573.302,Z 208.074,A -85,B 0,C 180,E1 -2162.811,E2 -2162.811} C_VEL
LIN {X 0,Y 573.296,Z 208.069,A -85,B 0,C 180,E1 -2165.628,E2 -2165.628} C_VEL
LIN {X 0,Y 573.282,Z 208.072,A -85,B 0,C 180,E1 -2168.46,E2 -2168.46} C_VEL
LIN {X 0,Y 573.269,Z 208.075,A -85,B 0,C 180,E1 -2171.312,E2 -2171.312} C_VEL
LIN {X 0,Y 573.279,Z 208.073,A -85,B 0,C 180,E1 -2174.425,E2 -2174.425} C_VEL
LIN {X 0,Y 573.256,Z 208.079,A -85,B 0,C 180,E1 -2177.112,E2 -2177.112} C_VEL
LIN {X 0,Y 573.25,Z 208.074,A -85,B 0,C 180,E1 -2180.077,E2 -2180.077} C_VEL
LIN {X 0,Y 573.232,Z 208.081,A -85,B 0,C 180,E1 -2183.1,E2 -2183.1} C_VEL
LIN {X 0,Y 573.25,Z 208.075,A -85,B 0,C 180,E1 -2185.41,E2 -2185.41} C_VEL
LIN {X 0,Y 573.25,Z 208.074,A -85,B 0,C 180,E1 -2188.029,E2 -2188.029} C_VEL
LIN {X 0,Y 573.244,Z 208.075,A -85,B 0,C 180,E1 -2190.176,E2 -2190.176} C_VEL
LIN {X 0,Y 573.251,Z 208.081,A -85,B 0,C 180,E1 -2192.645,E2 -2192.645} C_VEL
LIN {X 0,Y 573.253,Z 208.076,A -85,B 0,C 180,E1 -2195.185,E2 -2195.185} C_VEL
LIN {X 0,Y 573.234,Z 208.075,A -85,B 0,C 180,E1 -2197.808,E2 -2197.808} C_VEL
LIN {X 0,Y 573.243,Z 208.081,A -85,B 0,C 180,E1 -2200.525,E2 -2200.525} C_VEL
LIN {X 0,Y 573.237,Z 208.076,A -85,B 0,C 180,E1 -2203.359,E2 -2203.359} C_VEL
LIN {X 0,Y 573.246,Z 208.078,A -85,B 0,C 180,E1 -2206.331,E2 -2206.331} C_VEL
LIN {X 0,Y 573.229,Z 208.084,A -85,B 0,C 180,E1 -2208.543,E2 -2208.543} C_VEL
LIN {X 0,Y 573.238,Z 208.076,A -85,B 0,C 180,E1 -2211.298,E2 -2211.298} C_VEL
LIN {X 0,Y 573.193,Z 208.082,A -85,B 0,C 180,E1 -2214.022,E2 -2214.022} C_VEL
LIN {X 0,Y 573.27,Z 208.079,A -85,B 0,C 180,E1 -2216.518,E2 -2216.518} C_VEL
LIN {X 0,Y 573.225,Z 208.079,A -85,B 0,C 180,E1 -2219.119,E2 -2219.119} C_VEL
LIN {X 0,Y 573.23,Z 208.076,A -85,B 0,C 180,E1 -2221.435,E2 -2221.435} C_VEL
LIN {X 0,Y 573.236,Z 208.085,A -85,B 0,C 180,E1 -2224.589,E2 -2224.589} C_VEL
LIN {X 0,Y 573.237,Z 208.13,A -85,B 0,C 180,E1 -2226.968,E2 -2226.968} C_VEL
LIN {X 0,Y 573.955,Z 212.793,A -85,B 0,C 180,E1 -2227.692,E2 -2227.692} C_VEL
LIN {X 0,Y 573.783,Z 230.646,A -85,B 0,C 180,E1 -2230.317,E2 -2230.317} C_VEL
LIN {X 0,Y 573.542,Z 249.143,A -85,B 0,C 180,E1 -2233.023,E2 -2233.023} C_VEL
LIN {X 0,Y 573.401,Z 270.794,A -85,B 0,C 180,E1 -2236.15,E2 -2236.15} C_VEL
LIN {X 0,Y 574.061,Z 276.525,A -85,B 0,C 180,E1 -2236.256,E2 -2236.256} C_VEL
LIN {X 0,Y 573.877,Z 378.956,A -85,B 0,C 180,E1 -2237.558,E2 -2237.558} C_VEL
LIN {X 0,Y 573.785,Z 392.225,A -85,B 0,C 180,E1 -2237.87,E2 -2237.87} C_VEL
LIN {X 0,Y 573.676,Z 404.381,A -85,B 0,C 180,E1 -2238.294,E2 -2238.294} C_VEL
LIN {X 0,Y 573.602,Z 415.594,A -85,B 0,C 180,E1 -2238.818,E2 -2238.818} C_VEL
LIN {X 0,Y 573.478,Z 426.911,A -85,B 0,C 180,E1 -2239.497,E2 -2239.497} C_VEL
LIN {X 0,Y 573.349,Z 437.542,A -85,B 0,C 180,E1 -2240.297,E2 -2240.297} C_VEL
LIN {X 0,Y 573.241,Z 447.114,A -85,B 0,C 180,E1 -2241.185,E2 -2241.185} C_VEL
LIN {X 0,Y 573.161,Z 454.962,A -85,B 0,C 180,E1 -2242.071,E2 -2242.071} C_VEL
LIN {X 0,Y 573.072,Z 462.955,A -85,B 0,C 180,E1 -2243.185,E2 -2243.185} C_VEL
LIN {X 0,Y 573.07,Z 469.681,A -85,B 0,C 180,E1 -2244.37,E2 -2244.37} C_VEL
LIN {X 0,Y 573.028,Z 474.373,A -85,B 0,C 180,E1 -2245.428,E2 -2245.428} C_VEL
LIN {X 0,Y 573.022,Z 477.958,A -85,B 0,C 180,E1 -2246.484,E2 -2246.484} C_VEL
LIN {X 0,Y 572.959,Z 479.808,A -85,B 0,C 180,E1 -2247.188,E2 -2247.188} C_VEL
LIN {X 0,Y 572.946,Z 482.185,A -85,B 0,C 180,E1 -2248.594,E2 -2248.594} C_VEL
LIN {X 0,Y 572.938,Z 483,A -85,B 0,C 180,E1 -2250,E2 -2250} C_VEL
LIN {X 0,Y 572.946,Z 482.186,A -85,B 0,C 180,E1 -2251.406,E2 -2251.406} C_VEL
LIN {X 0,Y 572.939,Z 481.199,A -85,B 0,C 180,E1 -2252.109,E2 -2252.109} C_VEL
LIN {X 0,Y 572.959,Z 479.81,A -85,B 0,C 180,E1 -2252.812,E2 -2252.812} C_VEL
LIN {X 0,Y 573.015,Z 476.895,A -85,B 0,C 180,E1 -2253.868,E2 -2253.868} C_VEL
LIN {X 0,Y 572.963,Z 472.948,A -85,B 0,C 180,E1 -2254.926,E2 -2254.926} C_VEL
LIN {X 0,Y 573.064,Z 466.876,A -85,B 0,C 180,E1 -2256.16,E2 -2256.16} C_VEL
LIN {X 0,Y 573.119,Z 460.237,A -85,B 0,C 180,E1 -2257.221,E2 -2257.221} C_VEL
LIN {X 0,Y 573.201,Z 451.99,A -85,B 0,C 180,E1 -2258.283,E2 -2258.283} C_VEL
LIN {X 0,Y 573.287,Z 443.538,A -85,B 0,C 180,E1 -2259.17,E2 -2259.17} C_VEL
LIN {X 0,Y 573.424,Z 433.096,A -85,B 0,C 180,E1 -2260.058,E2 -2260.058} C_VEL
LIN {X 0,Y 573.555,Z 421.4,A -85,B 0,C 180,E1 -2260.855,E2 -2260.855} C_VEL
LIN {X 0,Y 573.653,Z 410.287,A -85,B 0,C 180,E1 -2261.447,E2 -2261.447} C_VEL
LIN {X 0,Y 573.725,Z 397.169,A -85,B 0,C 180,E1 -2261.975,E2 -2261.975} C_VEL
LIN {X 0,Y 573.84,Z 384.516,A -85,B 0,C 180,E1 -2262.331,E2 -2262.331} C_VEL
LIN {X 0,Y 573.891,Z 371.307,A -85,B 0,C 180,E1 -2262.555,E2 -2262.555} C_VEL
LIN {X 0,Y 573.878,Z 274.272,A -85,B 0,C 180,E1 -2263.777,E2 -2263.777} C_VEL
LIN {X 0,Y 573.4,Z 270.792,A -85,B 0,C 180,E1 -2263.85,E2 -2263.85} C_VEL
LIN {X 0,Y 573.536,Z 250.898,A -85,B 0,C 180,E1 -2266.722,E2 -2266.722} C_VEL
LIN {X 0,Y 573.732,Z 233.17,A -85,B 0,C 180,E1 -2269.314,E2 -2269.314} C_VEL
LIN {X 0,Y 573.937,Z 213.982,A -85,B 0,C 180,E1 -2272.12,E2 -2272.12} C_VEL
